Fanuc TP program (LS listing): hs_ov_h80_gutr.ls

/PROG  hs_ov_h80_gutr
/ATTR
COMMENT	= "19-03-05 13:35:50";
PROG_SIZE	= 0;
DEFAULT_GROUP	= 1, *, *, *, *;
/APPL
    ARC Welding Equipment: 1, *, *, *, *;
/MN
   1:  CALL HOME_ALL;
   1:  UFRAME_NUM = 1;
   1:  UTOOL_NUM = 3;
   1:  COL GUARD ADJUST 150;
   1:  PR[91] = PR[90];
   1:  PR[91,1] = PR[90,1] + 2.077;
   1:  PR[91,2] = PR[90,2] + 1.178;
   1:  PR[91,3] = PR[90,3] + 1.495;
   1:  PR[92] = PR[91];
   1:  PR[92,3] = PR[92,3] + 50;
   1:J PR[92] 10% FINE;
   1:L PR[91] R[100]mm/sec CNT100;
   1:  CALL LASER_DRAHT_START;
   1:  PR[91,1] = PR[90,1] + -2.557;
   1:L PR[91] R[100]mm/sec CNT100;
   1:  PR[91,1] = PR[90,1] + -4.760;
   1:  PR[91,2] = PR[90,2] + 1.925;
   1:L PR[91] R[100]mm/sec CNT100;
   1:  PR[91,1] = PR[90,1] + -5.957;
   1:  PR[91,2] = PR[90,2] + 3.712;
   1:L PR[91] R[100]mm/sec CNT100;
   1:  PR[91,1] = PR[90,1] + -7.859;
   1:  PR[91,2] = PR[90,2] + 8.118;
   1:L PR[91] R[100]mm/sec CNT100;
   1:  PR[91,1] = PR[90,1] + -8.020;
   1:  PR[91,2] = PR[90,2] + 8.503;
   1:L PR[91] R[100]mm/sec CNT100;
   1:  PR[91,1] = PR[90,1] + -8.141;
   1:  PR[91,2] = PR[90,2] + 8.842;
   1:L PR[91] R[100]mm/sec CNT100;
   1:  PR[91,1] = PR[90,1] + -8.162;
   1:  PR[91,2] = PR[90,2] + 8.883;
   1:L PR[91] R[100]mm/sec CNT100;
   1:  PR[91,1] = PR[90,1] + -11.179;
   1:  PR[91,2] = PR[90,2] + 12.501;
   1:L PR[91] R[100]mm/sec CNT100;
   1:  PR[91,1] = PR[90,1] + -11.400;
   1:  PR[91,2] = PR[90,2] + 12.803;
   1:L PR[91] R[100]mm/sec CNT100;
   1:  PR[91,1] = PR[90,1] + -11.431;
   1:  PR[91,2] = PR[90,2] + 12.835;
   1:L PR[91] R[100]mm/sec CNT100;
   1:  PR[91,1] = PR[90,1] + -15.350;
   1:  PR[91,2] = PR[90,2] + 15.448;
   1:L PR[91] R[100]mm/sec CNT100;
   1:  PR[91,1] = PR[90,1] + -15.648;
   1:  PR[91,2] = PR[90,2] + 15.676;
   1:L PR[91] R[100]mm/sec CNT100;
   1:  PR[91,1] = PR[90,1] + -15.686;
   1:  PR[91,2] = PR[90,2] + 15.697;
   1:L PR[91] R[100]mm/sec CNT100;
   1:  PR[91,1] = PR[90,1] + -20.186;
   1:  PR[91,2] = PR[90,2] + 17.090;
   1:L PR[91] R[100]mm/sec CNT100;
   1:  PR[91,1] = PR[90,1] + -20.537;
   1:  PR[91,2] = PR[90,2] + 17.225;
   1:L PR[91] R[100]mm/sec CNT100;
   1:  PR[91,1] = PR[90,1] + -20.579;
   1:  PR[91,2] = PR[90,2] + 17.235;
   1:L PR[91] R[100]mm/sec CNT100;
   1:  PR[91,1] = PR[90,1] + -25.291;
   1:  PR[91,2] = PR[90,2] + 17.293;
   1:L PR[91] R[100]mm/sec CNT100;
   1:  PR[91,1] = PR[90,1] + -25.667;
   1:  PR[91,2] = PR[90,2] + 17.323;
   1:L PR[91] R[100]mm/sec CNT100;
   1:  PR[91,1] = PR[90,1] + -25.709;
   1:  PR[91,2] = PR[90,2] + 17.320;
   1:L PR[91] R[100]mm/sec CNT100;
   1:  PR[91,1] = PR[90,1] + -30.244;
   1:  PR[91,2] = PR[90,2] + 16.038;
   1:L PR[91] R[100]mm/sec CNT100;
   1:  PR[91,1] = PR[90,1] + -30.614;
   1:  PR[91,2] = PR[90,2] + 15.960;
   1:L PR[91] R[100]mm/sec CNT100;
   1:  PR[91,1] = PR[90,1] + -30.652;
   1:  PR[91,2] = PR[90,2] + 15.946;
   1:L PR[91] R[100]mm/sec CNT100;
   1:  PR[91,1] = PR[90,1] + -34.635;
   1:  PR[91,2] = PR[90,2] + 13.430;
   1:L PR[91] R[100]mm/sec CNT100;
   1:  PR[91,1] = PR[90,1] + -34.968;
   1:  PR[91,2] = PR[90,2] + 13.250;
   1:L PR[91] R[100]mm/sec CNT100;
   1:  PR[91,1] = PR[90,1] + -35.000;
   1:  PR[91,2] = PR[90,2] + 13.227;
   1:L PR[91] R[100]mm/sec CNT100;
   1:  PR[91,1] = PR[90,1] + -38.105;
   1:  PR[91,2] = PR[90,2] + 9.684;
   1:L PR[91] R[100]mm/sec CNT100;
   1:  PR[91,1] = PR[90,1] + -38.375;
   1:  PR[91,2] = PR[90,2] + 9.416;
   1:L PR[91] R[100]mm/sec CNT100;
   1:  PR[91,1] = PR[90,1] + -38.398;
   1:  PR[91,2] = PR[90,2] + 9.386;
   1:L PR[91] R[100]mm/sec CNT100;
   1:  PR[91,1] = PR[90,1] + -40.370;
   1:  PR[91,2] = PR[90,2] + 5.107;
   1:L PR[91] R[100]mm/sec CNT100;
   1:  PR[91,1] = PR[90,1] + -40.554;
   1:  PR[91,2] = PR[90,2] + 4.773;
   1:L PR[91] R[100]mm/sec CNT100;
   1:  PR[91,1] = PR[90,1] + -40.567;
   1:  PR[91,2] = PR[90,2] + 4.738;
   1:L PR[91] R[100]mm/sec CNT100;
   1:  PR[91,1] = PR[90,1] + -41.243;
   1:  PR[91,2] = PR[90,2] + 0.073;
   1:L PR[91] R[100]mm/sec CNT100;
   1:  PR[91,1] = PR[90,1] + -41.325;
   1:  PR[91,2] = PR[90,2] + -0.300;
   1:L PR[91] R[100]mm/sec CNT100;
   1:  PR[91,1] = PR[90,1] + -41.327;
   1:  PR[91,2] = PR[90,2] + -0.336;
   1:L PR[91] R[100]mm/sec CNT100;
   1:  PR[91,1] = PR[90,1] + -40.651;
   1:  PR[91,2] = PR[90,2] + -5.001;
   1:L PR[91] R[100]mm/sec CNT100;
   1:  PR[91,1] = PR[90,1] + -40.624;
   1:  PR[91,2] = PR[90,2] + -5.383;
   1:L PR[91] R[100]mm/sec CNT100;
   1:  PR[91,1] = PR[90,1] + -40.597;
   1:  PR[91,2] = PR[90,2] + -5.504;
   1:L PR[91] R[100]mm/sec CNT100;
   1:  PR[91,1] = PR[90,1] + -40.524;
   1:  PR[91,2] = PR[90,2] + -5.699;
   1:L PR[91] R[100]mm/sec CNT100;
   1:  PR[91,1] = PR[90,1] + -38.552;
   1:  PR[91,2] = PR[90,2] + -9.979;
   1:L PR[91] R[100]mm/sec CNT100;
   1:  PR[91,1] = PR[90,1] + -38.450;
   1:  PR[91,2] = PR[90,2] + -10.165;
   1:L PR[91] R[100]mm/sec CNT100;
   1:  PR[91,1] = PR[90,1] + -38.325;
   1:  PR[91,2] = PR[90,2] + -10.331;
   1:L PR[91] R[100]mm/sec CNT100;
   1:  PR[91,1] = PR[90,1] + -35.219;
   1:  PR[91,2] = PR[90,2] + -13.874;
   1:L PR[91] R[100]mm/sec CNT100;
   1:  PR[91,1] = PR[90,1] + -35.068;
   1:  PR[91,2] = PR[90,2] + -14.024;
   1:L PR[91] R[100]mm/sec CNT100;
   1:  PR[91,1] = PR[90,1] + -34.902;
   1:  PR[91,2] = PR[90,2] + -14.147;
   1:L PR[91] R[100]mm/sec CNT100;
   1:  PR[91,1] = PR[90,1] + -30.918;
   1:  PR[91,2] = PR[90,2] + -16.664;
   1:L PR[91] R[100]mm/sec CNT100;
   1:  PR[91,1] = PR[90,1] + -30.730;
   1:  PR[91,2] = PR[90,2] + -16.765;
   1:L PR[91] R[100]mm/sec CNT100;
   1:  PR[91,1] = PR[90,1] + -30.537;
   1:  PR[91,2] = PR[90,2] + -16.836;
   1:L PR[91] R[100]mm/sec CNT100;
   1:  PR[91,1] = PR[90,1] + -26.001;
   1:  PR[91,2] = PR[90,2] + -18.118;
   1:L PR[91] R[100]mm/sec CNT100;
   1:  PR[91,1] = PR[90,1] + -25.791;
   1:  PR[91,2] = PR[90,2] + -18.162;
   1:L PR[91] R[100]mm/sec CNT100;
   1:  PR[91,1] = PR[90,1] + -25.587;
   1:  PR[91,2] = PR[90,2] + -18.175;
   1:L PR[91] R[100]mm/sec CNT100;
   1:  PR[91,1] = PR[90,1] + -20.873;
   1:  PR[91,2] = PR[90,2] + -18.117;
   1:L PR[91] R[100]mm/sec CNT100;
   1:  PR[91,1] = PR[90,1] + -20.658;
   1:  PR[91,2] = PR[90,2] + -18.100;
   1:L PR[91] R[100]mm/sec CNT100;
   1:  PR[91,1] = PR[90,1] + -20.460;
   1:  PR[91,2] = PR[90,2] + -18.055;
   1:L PR[91] R[100]mm/sec CNT100;
   1:  PR[91,1] = PR[90,1] + -15.959;
   1:  PR[91,2] = PR[90,2] + -16.661;
   1:L PR[91] R[100]mm/sec CNT100;
   1:  PR[91,1] = PR[90,1] + -15.756;
   1:  PR[91,2] = PR[90,2] + -16.583;
   1:L PR[91] R[100]mm/sec CNT100;
   1:  PR[91,1] = PR[90,1] + -15.579;
   1:  PR[91,2] = PR[90,2] + -16.484;
   1:L PR[91] R[100]mm/sec CNT100;
   1:  PR[91,1] = PR[90,1] + -11.659;
   1:  PR[91,2] = PR[90,2] + -13.871;
   1:L PR[91] R[100]mm/sec CNT100;
   1:  PR[91,1] = PR[90,1] + -11.486;
   1:  PR[91,2] = PR[90,2] + -13.739;
   1:L PR[91] R[100]mm/sec CNT100;
   1:  PR[91,1] = PR[90,1] + -11.345;
   1:  PR[91,2] = PR[90,2] + -13.595;
   1:L PR[91] R[100]mm/sec CNT100;
   1:  PR[91,1] = PR[90,1] + -8.328;
   1:  PR[91,2] = PR[90,2] + -9.976;
   1:L PR[91] R[100]mm/sec CNT100;
   1:  PR[91,1] = PR[90,1] + -8.199;
   1:  PR[91,2] = PR[90,2] + -9.799;
   1:L PR[91] R[100]mm/sec CNT100;
   1:  PR[91,1] = PR[90,1] + -8.105;
   1:  PR[91,2] = PR[90,2] + -9.621;
   1:L PR[91] R[100]mm/sec CNT100;
   1:  PR[91,1] = PR[90,1] + -6.242;
   1:  PR[91,2] = PR[90,2] + -5.303;
   1:L PR[91] R[100]mm/sec CNT100;
   1:  PR[91,1] = PR[90,1] + -6.003;
   1:  PR[91,2] = PR[90,2] + -4.628;
   1:L PR[91] R[100]mm/sec CNT100;
   1:  PR[91,1] = PR[90,1] + -4.760;
   1:  PR[91,2] = PR[90,2] + -2.773;
   1:L PR[91] R[100]mm/sec CNT100;
   1:  PR[91,1] = PR[90,1] + -2.557;
   1:  PR[91,2] = PR[90,2] + -2.026;
   1:L PR[91] R[100]mm/sec CNT100;
   1:  PR[91,1] = PR[90,1] + 2.077;
   1:L PR[91] R[100]mm/sec CNT100;
   1:  PR[91,1] = PR[90,1] + 4.281;
   1:  PR[91,2] = PR[90,2] + -2.773;
   1:L PR[91] R[100]mm/sec CNT100;
   1:  PR[91,1] = PR[90,1] + 5.478;
   1:  PR[91,2] = PR[90,2] + -4.559;
   1:L PR[91] R[100]mm/sec CNT100;
   1:  PR[91,1] = PR[90,1] + 7.379;
   1:  PR[91,2] = PR[90,2] + -8.965;
   1:L PR[91] R[100]mm/sec CNT100;
   1:  PR[91,1] = PR[90,1] + 7.540;
   1:  PR[91,2] = PR[90,2] + -9.350;
   1:L PR[91] R[100]mm/sec CNT100;
   1:  PR[91,1] = PR[90,1] + 7.661;
   1:  PR[91,2] = PR[90,2] + -9.690;
   1:L PR[91] R[100]mm/sec CNT100;
   1:  PR[91,1] = PR[90,1] + 7.683;
   1:  PR[91,2] = PR[90,2] + -9.730;
   1:L PR[91] R[100]mm/sec CNT100;
   1:  PR[91,1] = PR[90,1] + 10.700;
   1:  PR[91,2] = PR[90,2] + -13.348;
   1:L PR[91] R[100]mm/sec CNT100;
   1:  PR[91,1] = PR[90,1] + 10.920;
   1:  PR[91,2] = PR[90,2] + -13.650;
   1:L PR[91] R[100]mm/sec CNT100;
   1:  PR[91,1] = PR[90,1] + 10.951;
   1:  PR[91,2] = PR[90,2] + -13.682;
   1:L PR[91] R[100]mm/sec CNT100;
   1:  PR[91,1] = PR[90,1] + 14.871;
   1:  PR[91,2] = PR[90,2] + -16.295;
   1:L PR[91] R[100]mm/sec CNT100;
   1:  PR[91,1] = PR[90,1] + 15.168;
   1:  PR[91,2] = PR[90,2] + -16.523;
   1:L PR[91] R[100]mm/sec CNT100;
   1:  PR[91,1] = PR[90,1] + 15.207;
   1:  PR[91,2] = PR[90,2] + -16.544;
   1:L PR[91] R[100]mm/sec CNT100;
   1:  PR[91,1] = PR[90,1] + 19.707;
   1:  PR[91,2] = PR[90,2] + -17.938;
   1:L PR[91] R[100]mm/sec CNT100;
   1:  PR[91,1] = PR[90,1] + 20.058;
   1:  PR[91,2] = PR[90,2] + -18.072;
   1:L PR[91] R[100]mm/sec CNT100;
   1:  PR[91,1] = PR[90,1] + 20.099;
   1:  PR[91,2] = PR[90,2] + -18.082;
   1:L PR[91] R[100]mm/sec CNT100;
   1:  PR[91,1] = PR[90,1] + 24.812;
   1:  PR[91,2] = PR[90,2] + -18.140;
   1:L PR[91] R[100]mm/sec CNT100;
   1:  PR[91,1] = PR[90,1] + 25.187;
   1:  PR[91,2] = PR[90,2] + -18.170;
   1:L PR[91] R[100]mm/sec CNT100;
   1:  PR[91,1] = PR[90,1] + 25.229;
   1:  PR[91,2] = PR[90,2] + -18.168;
   1:L PR[91] R[100]mm/sec CNT100;
   1:  PR[91,1] = PR[90,1] + 29.764;
   1:  PR[91,2] = PR[90,2] + -16.885;
   1:L PR[91] R[100]mm/sec CNT100;
   1:  PR[91,1] = PR[90,1] + 30.134;
   1:  PR[91,2] = PR[90,2] + -16.808;
   1:L PR[91] R[100]mm/sec CNT100;
   1:  PR[91,1] = PR[90,1] + 30.172;
   1:  PR[91,2] = PR[90,2] + -16.794;
   1:L PR[91] R[100]mm/sec CNT100;
   1:  PR[91,1] = PR[90,1] + 34.155;
   1:  PR[91,2] = PR[90,2] + -14.277;
   1:L PR[91] R[100]mm/sec CNT100;
   1:  PR[91,1] = PR[90,1] + 34.489;
   1:  PR[91,2] = PR[90,2] + -14.098;
   1:L PR[91] R[100]mm/sec CNT100;
   1:  PR[91,1] = PR[90,1] + 34.521;
   1:  PR[91,2] = PR[90,2] + -14.074;
   1:L PR[91] R[100]mm/sec CNT100;
   1:  PR[91,1] = PR[90,1] + 37.626;
   1:  PR[91,2] = PR[90,2] + -10.531;
   1:L PR[91] R[100]mm/sec CNT100;
   1:  PR[91,1] = PR[90,1] + 37.895;
   1:  PR[91,2] = PR[90,2] + -10.264;
   1:L PR[91] R[100]mm/sec CNT100;
   1:  PR[91,1] = PR[90,1] + 37.919;
   1:  PR[91,2] = PR[90,2] + -10.233;
   1:L PR[91] R[100]mm/sec CNT100;
   1:  PR[91,1] = PR[90,1] + 39.891;
   1:  PR[91,2] = PR[90,2] + -5.954;
   1:L PR[91] R[100]mm/sec CNT100;
   1:  PR[91,1] = PR[90,1] + 40.074;
   1:  PR[91,2] = PR[90,2] + -5.620;
   1:L PR[91] R[100]mm/sec CNT100;
   1:  PR[91,1] = PR[90,1] + 40.087;
   1:  PR[91,2] = PR[90,2] + -5.585;
   1:L PR[91] R[100]mm/sec CNT100;
   1:  PR[91,1] = PR[90,1] + 40.764;
   1:  PR[91,2] = PR[90,2] + -0.920;
   1:L PR[91] R[100]mm/sec CNT100;
   1:  PR[91,1] = PR[90,1] + 40.845;
   1:  PR[91,2] = PR[90,2] + -0.547;
   1:L PR[91] R[100]mm/sec CNT100;
   1:  PR[91,1] = PR[90,1] + 40.848;
   1:  PR[91,2] = PR[90,2] + -0.511;
   1:L PR[91] R[100]mm/sec CNT100;
   1:  PR[91,1] = PR[90,1] + 40.171;
   1:  PR[91,2] = PR[90,2] + 4.154;
   1:L PR[91] R[100]mm/sec CNT100;
   1:  PR[91,1] = PR[90,1] + 40.144;
   1:  PR[91,2] = PR[90,2] + 4.536;
   1:L PR[91] R[100]mm/sec CNT100;
   1:  PR[91,1] = PR[90,1] + 40.117;
   1:  PR[91,2] = PR[90,2] + 4.657;
   1:L PR[91] R[100]mm/sec CNT100;
   1:  PR[91,1] = PR[90,1] + 40.044;
   1:  PR[91,2] = PR[90,2] + 4.852;
   1:L PR[91] R[100]mm/sec CNT100;
   1:  PR[91,1] = PR[90,1] + 38.072;
   1:  PR[91,2] = PR[90,2] + 9.132;
   1:L PR[91] R[100]mm/sec CNT100;
   1:  PR[91,1] = PR[90,1] + 37.970;
   1:  PR[91,2] = PR[90,2] + 9.318;
   1:L PR[91] R[100]mm/sec CNT100;
   1:  PR[91,1] = PR[90,1] + 37.845;
   1:  PR[91,2] = PR[90,2] + 9.483;
   1:L PR[91] R[100]mm/sec CNT100;
   1:  PR[91,1] = PR[90,1] + 34.739;
   1:  PR[91,2] = PR[90,2] + 13.027;
   1:L PR[91] R[100]mm/sec CNT100;
   1:  PR[91,1] = PR[90,1] + 34.588;
   1:  PR[91,2] = PR[90,2] + 13.177;
   1:L PR[91] R[100]mm/sec CNT100;
   1:  PR[91,1] = PR[90,1] + 34.422;
   1:  PR[91,2] = PR[90,2] + 13.300;
   1:L PR[91] R[100]mm/sec CNT100;
   1:  PR[91,1] = PR[90,1] + 30.438;
   1:  PR[91,2] = PR[90,2] + 15.816;
   1:L PR[91] R[100]mm/sec CNT100;
   1:  PR[91,1] = PR[90,1] + 30.250;
   1:  PR[91,2] = PR[90,2] + 15.918;
   1:L PR[91] R[100]mm/sec CNT100;
   1:  PR[91,1] = PR[90,1] + 30.057;
   1:  PR[91,2] = PR[90,2] + 15.988;
   1:L PR[91] R[100]mm/sec CNT100;
   1:  PR[91,1] = PR[90,1] + 25.521;
   1:  PR[91,2] = PR[90,2] + 17.271;
   1:L PR[91] R[100]mm/sec CNT100;
   1:  PR[91,1] = PR[90,1] + 25.311;
   1:  PR[91,2] = PR[90,2] + 17.315;
   1:L PR[91] R[100]mm/sec CNT100;
   1:  PR[91,1] = PR[90,1] + 25.107;
   1:  PR[91,2] = PR[90,2] + 17.328;
   1:L PR[91] R[100]mm/sec CNT100;
   1:  PR[91,1] = PR[90,1] + 20.394;
   1:  PR[91,2] = PR[90,2] + 17.270;
   1:L PR[91] R[100]mm/sec CNT100;
   1:  PR[91,1] = PR[90,1] + 20.178;
   1:  PR[91,2] = PR[90,2] + 17.253;
   1:L PR[91] R[100]mm/sec CNT100;
   1:  PR[91,1] = PR[90,1] + 19.980;
   1:  PR[91,2] = PR[90,2] + 17.207;
   1:L PR[91] R[100]mm/sec CNT100;
   1:  PR[91,1] = PR[90,1] + 15.479;
   1:  PR[91,2] = PR[90,2] + 15.814;
   1:L PR[91] R[100]mm/sec CNT100;
   1:  PR[91,1] = PR[90,1] + 15.276;
   1:  PR[91,2] = PR[90,2] + 15.736;
   1:L PR[91] R[100]mm/sec CNT100;
   1:  PR[91,1] = PR[90,1] + 15.100;
   1:  PR[91,2] = PR[90,2] + 15.637;
   1:L PR[91] R[100]mm/sec CNT100;
   1:  PR[91,1] = PR[90,1] + 11.180;
   1:  PR[91,2] = PR[90,2] + 13.024;
   1:L PR[91] R[100]mm/sec CNT100;
   1:  PR[91,1] = PR[90,1] + 11.007;
   1:  PR[91,2] = PR[90,2] + 12.892;
   1:L PR[91] R[100]mm/sec CNT100;
   1:  PR[91,1] = PR[90,1] + 10.866;
   1:  PR[91,2] = PR[90,2] + 12.747;
   1:L PR[91] R[100]mm/sec CNT100;
   1:  PR[91,1] = PR[90,1] + 7.848;
   1:  PR[91,2] = PR[90,2] + 9.129;
   1:L PR[91] R[100]mm/sec CNT100;
   1:  PR[91,1] = PR[90,1] + 7.719;
   1:  PR[91,2] = PR[90,2] + 8.952;
   1:L PR[91] R[100]mm/sec CNT100;
   1:  PR[91,1] = PR[90,1] + 7.625;
   1:  PR[91,2] = PR[90,2] + 8.774;
   1:L PR[91] R[100]mm/sec CNT100;
   1:  PR[91,1] = PR[90,1] + 5.762;
   1:  PR[91,2] = PR[90,2] + 4.456;
   1:L PR[91] R[100]mm/sec CNT100;
   1:  PR[91,1] = PR[90,1] + 5.524;
   1:  PR[91,2] = PR[90,2] + 3.781;
   1:L PR[91] R[100]mm/sec CNT100;
   1:  PR[91,1] = PR[90,1] + 4.281;
   1:  PR[91,2] = PR[90,2] + 1.925;
   1:L PR[91] R[100]mm/sec CNT100;
   1:  PR[91,1] = PR[90,1] + 2.077;
   1:  PR[91,2] = PR[90,2] + 1.178;
   1:L PR[91] R[100]mm/sec CNT100;
   1:  PR[91] = PR[90];
   1:  PR[91,1] = PR[90,1] + -2.557;
   1:  PR[91,3] = PR[90,3] + 2.795;
   1:L PR[91] R[100]mm/sec CNT100;
   1:  PR[91,1] = PR[90,1] + -4.760;
   1:  PR[91,2] = PR[90,2] + 1.925;
   1:L PR[91] R[100]mm/sec CNT100;
   1:  PR[91,1] = PR[90,1] + -5.959;
   1:  PR[91,2] = PR[90,2] + 3.715;
   1:L PR[91] R[100]mm/sec CNT100;
   1:  PR[91,1] = PR[90,1] + -7.336;
   1:  PR[91,2] = PR[90,2] + 6.933;
   1:L PR[91] R[100]mm/sec CNT100;
   1:  PR[91,1] = PR[90,1] + -7.755;
   1:  PR[91,2] = PR[90,2] + 8.106;
   1:L PR[91] R[100]mm/sec CNT100;
   1:  PR[91,1] = PR[90,1] + -8.186;
   1:  PR[91,2] = PR[90,2] + 8.922;
   1:L PR[91] R[100]mm/sec CNT100;
   1:  PR[91,1] = PR[90,1] + -10.080;
   1:  PR[91,2] = PR[90,2] + 11.193;
   1:L PR[91] R[100]mm/sec CNT100;
   1:  PR[91,1] = PR[90,1] + -10.818;
   1:  PR[91,2] = PR[90,2] + 12.203;
   1:L PR[91] R[100]mm/sec CNT100;
   1:  PR[91,1] = PR[90,1] + -11.462;
   1:  PR[91,2] = PR[90,2] + 12.862;
   1:L PR[91] R[100]mm/sec CNT100;
   1:  PR[91,1] = PR[90,1] + -13.922;
   1:  PR[91,2] = PR[90,2] + 14.503;
   1:L PR[91] R[100]mm/sec CNT100;
   1:  PR[91,1] = PR[90,1] + -14.916;
   1:  PR[91,2] = PR[90,2] + 15.263;
   1:L PR[91] R[100]mm/sec CNT100;
   1:  PR[91,1] = PR[90,1] + -15.719;
   1:  PR[91,2] = PR[90,2] + 15.713;
   1:L PR[91] R[100]mm/sec CNT100;
   1:  PR[91,1] = PR[90,1] + -18.544;
   1:  PR[91,2] = PR[90,2] + 16.587;
   1:L PR[91] R[100]mm/sec CNT100;
   1:  PR[91,1] = PR[90,1] + -19.713;
   1:  PR[91,2] = PR[90,2] + 17.036;
   1:L PR[91] R[100]mm/sec CNT100;
   1:  PR[91,1] = PR[90,1] + -20.610;
   1:  PR[91,2] = PR[90,2] + 17.239;
   1:L PR[91] R[100]mm/sec CNT100;
   1:  PR[91,1] = PR[90,1] + -23.569;
   1:  PR[91,2] = PR[90,2] + 17.276;
   1:L PR[91] R[100]mm/sec CNT100;
   1:  PR[91,1] = PR[90,1] + -24.818;
   1:  PR[91,2] = PR[90,2] + 17.376;
   1:L PR[91] R[100]mm/sec CNT100;
   1:  PR[91,1] = PR[90,1] + -25.734;
   1:  PR[91,2] = PR[90,2] + 17.317;
   1:L PR[91] R[100]mm/sec CNT100;
   1:  PR[91,1] = PR[90,1] + -28.581;
   1:  PR[91,2] = PR[90,2] + 16.512;
   1:L PR[91] R[100]mm/sec CNT100;
   1:  PR[91,1] = PR[90,1] + -29.809;
   1:  PR[91,2] = PR[90,2] + 16.253;
   1:L PR[91] R[100]mm/sec CNT100;
   1:  PR[91,1] = PR[90,1] + -30.670;
   1:  PR[91,2] = PR[90,2] + 15.938;
   1:L PR[91] R[100]mm/sec CNT100;
   1:  PR[91,1] = PR[90,1] + -33.171;
   1:  PR[91,2] = PR[90,2] + 14.358;
   1:L PR[91] R[100]mm/sec CNT100;
   1:  PR[91,1] = PR[90,1] + -34.276;
   1:  PR[91,2] = PR[90,2] + 13.762;
   1:L PR[91] R[100]mm/sec CNT100;
   1:  PR[91,1] = PR[90,1] + -35.012;
   1:  PR[91,2] = PR[90,2] + 13.217;
   1:L PR[91] R[100]mm/sec CNT100;
   1:  PR[91,1] = PR[90,1] + -36.961;
   1:  PR[91,2] = PR[90,2] + 10.993;
   1:L PR[91] R[100]mm/sec CNT100;
   1:  PR[91,1] = PR[90,1] + -37.853;
   1:  PR[91,2] = PR[90,2] + 10.108;
   1:L PR[91] R[100]mm/sec CNT100;
   1:  PR[91,1] = PR[90,1] + -38.404;
   1:  PR[91,2] = PR[90,2] + 9.377;
   1:L PR[91] R[100]mm/sec CNT100;
   1:  PR[91,1] = PR[90,1] + -39.642;
   1:  PR[91,2] = PR[90,2] + 6.690;
   1:L PR[91] R[100]mm/sec CNT100;
   1:  PR[91,1] = PR[90,1] + -40.248;
   1:  PR[91,2] = PR[90,2] + 5.588;
   1:L PR[91] R[100]mm/sec CNT100;
   1:  PR[91,1] = PR[90,1] + -40.569;
   1:  PR[91,2] = PR[90,2] + 4.732;
   1:L PR[91] R[100]mm/sec CNT100;
   1:  PR[91,1] = PR[90,1] + -40.993;
   1:  PR[91,2] = PR[90,2] + 1.804;
   1:L PR[91] R[100]mm/sec CNT100;
   1:  PR[91,1] = PR[90,1] + -41.262;
   1:  PR[91,2] = PR[90,2] + 0.574;
   1:L PR[91] R[100]mm/sec CNT100;
   1:  PR[91,1] = PR[90,1] + -41.327;
   1:  PR[91,2] = PR[90,2] + -0.336;
   1:L PR[91] R[100]mm/sec CNT100;
   1:  PR[91,1] = PR[90,1] + -40.903;
   1:  PR[91,2] = PR[90,2] + -3.265;
   1:L PR[91] R[100]mm/sec CNT100;
   1:  PR[91,1] = PR[90,1] + -40.812;
   1:  PR[91,2] = PR[90,2] + -4.521;
   1:L PR[91] R[100]mm/sec CNT100;
   1:  PR[91,1] = PR[90,1] + -40.599;
   1:  PR[91,2] = PR[90,2] + -5.499;
   1:L PR[91] R[100]mm/sec CNT100;
   1:  PR[91,1] = PR[90,1] + -40.218;
   1:  PR[91,2] = PR[90,2] + -6.515;
   1:L PR[91] R[100]mm/sec CNT100;
   1:  PR[91,1] = PR[90,1] + -38.979;
   1:  PR[91,2] = PR[90,2] + -9.202;
   1:L PR[91] R[100]mm/sec CNT100;
   1:  PR[91,1] = PR[90,1] + -38.455;
   1:  PR[91,2] = PR[90,2] + -10.156;
   1:L PR[91] R[100]mm/sec CNT100;
   1:  PR[91,1] = PR[90,1] + -37.803;
   1:  PR[91,2] = PR[90,2] + -11.022;
   1:L PR[91] R[100]mm/sec CNT100;
   1:  PR[91,1] = PR[90,1] + -35.853;
   1:  PR[91,2] = PR[90,2] + -13.246;
   1:L PR[91] R[100]mm/sec CNT100;
   1:  PR[91,1] = PR[90,1] + -35.080;
   1:  PR[91,2] = PR[90,2] + -14.014;
   1:L PR[91] R[100]mm/sec CNT100;
   1:  PR[91,1] = PR[90,1] + -34.210;
   1:  PR[91,2] = PR[90,2] + -14.659;
   1:L PR[91] R[100]mm/sec CNT100;
   1:  PR[91,1] = PR[90,1] + -31.708;
   1:  PR[91,2] = PR[90,2] + -16.239;
   1:L PR[91] R[100]mm/sec CNT100;
   1:  PR[91,1] = PR[90,1] + -30.749;
   1:  PR[91,2] = PR[90,2] + -16.757;
   1:L PR[91] R[100]mm/sec CNT100;
   1:  PR[91,1] = PR[90,1] + -29.732;
   1:  PR[91,2] = PR[90,2] + -17.129;
   1:L PR[91] R[100]mm/sec CNT100;
   1:  PR[91,1] = PR[90,1] + -26.884;
   1:  PR[91,2] = PR[90,2] + -17.934;
   1:L PR[91] R[100]mm/sec CNT100;
   1:  PR[91,1] = PR[90,1] + -25.817;
   1:  PR[91,2] = PR[90,2] + -18.159;
   1:L PR[91] R[100]mm/sec CNT100;
   1:  PR[91,1] = PR[90,1] + -24.738;
   1:  PR[91,2] = PR[90,2] + -18.228;
   1:L PR[91] R[100]mm/sec CNT100;
   1:  PR[91,1] = PR[90,1] + -21.778;
   1:  PR[91,2] = PR[90,2] + -18.191;
   1:L PR[91] R[100]mm/sec CNT100;
   1:  PR[91,1] = PR[90,1] + -20.689;
   1:  PR[91,2] = PR[90,2] + -18.105;
   1:L PR[91] R[100]mm/sec CNT100;
   1:  PR[91,1] = PR[90,1] + -19.636;
   1:  PR[91,2] = PR[90,2] + -17.866;
   1:L PR[91] R[100]mm/sec CNT100;
   1:  PR[91,1] = PR[90,1] + -16.810;
   1:  PR[91,2] = PR[90,2] + -16.991;
   1:L PR[91] R[100]mm/sec CNT100;
   1:  PR[91,1] = PR[90,1] + -15.789;
   1:  PR[91,2] = PR[90,2] + -16.599;
   1:L PR[91] R[100]mm/sec CNT100;
   1:  PR[91,1] = PR[90,1] + -14.847;
   1:  PR[91,2] = PR[90,2] + -16.072;
   1:L PR[91] R[100]mm/sec CNT100;
   1:  PR[91,1] = PR[90,1] + -12.386;
   1:  PR[91,2] = PR[90,2] + -14.431;
   1:L PR[91] R[100]mm/sec CNT100;
   1:  PR[91,1] = PR[90,1] + -11.517;
   1:  PR[91,2] = PR[90,2] + -13.766;
   1:L PR[91] R[100]mm/sec CNT100;
   1:  PR[91,1] = PR[90,1] + -10.763;
   1:  PR[91,2] = PR[90,2] + -12.995;
   1:L PR[91] R[100]mm/sec CNT100;
   1:  PR[91,1] = PR[90,1] + -8.869;
   1:  PR[91,2] = PR[90,2] + -10.723;
   1:L PR[91] R[100]mm/sec CNT100;
   1:  PR[91,1] = PR[90,1] + -8.223;
   1:  PR[91,2] = PR[90,2] + -9.838;
   1:L PR[91] R[100]mm/sec CNT100;
   1:  PR[91,1] = PR[90,1] + -7.719;
   1:  PR[91,2] = PR[90,2] + -8.886;
   1:L PR[91] R[100]mm/sec CNT100;
   1:  PR[91,1] = PR[90,1] + -6.550;
   1:  PR[91,2] = PR[90,2] + -6.176;
   1:L PR[91] R[100]mm/sec CNT100;
   1:  PR[91,1] = PR[90,1] + -6.003;
   1:  PR[91,2] = PR[90,2] + -4.628;
   1:L PR[91] R[100]mm/sec CNT100;
   1:  PR[91,1] = PR[90,1] + -4.760;
   1:  PR[91,2] = PR[90,2] + -2.773;
   1:L PR[91] R[100]mm/sec CNT100;
   1:  PR[91,1] = PR[90,1] + -2.557;
   1:  PR[91,2] = PR[90,2] + -2.026;
   1:L PR[91] R[100]mm/sec CNT100;
   1:  PR[91,1] = PR[90,1] + 2.077;
   1:L PR[91] R[100]mm/sec CNT100;
   1:  PR[91,1] = PR[90,1] + 4.280;
   1:  PR[91,2] = PR[90,2] + -2.773;
   1:L PR[91] R[100]mm/sec CNT100;
   1:  PR[91,1] = PR[90,1] + 5.480;
   1:  PR[91,2] = PR[90,2] + -4.563;
   1:L PR[91] R[100]mm/sec CNT100;
   1:  PR[91,1] = PR[90,1] + 6.856;
   1:  PR[91,2] = PR[90,2] + -7.781;
   1:L PR[91] R[100]mm/sec CNT100;
   1:  PR[91,1] = PR[90,1] + 7.275;
   1:  PR[91,2] = PR[90,2] + -8.954;
   1:L PR[91] R[100]mm/sec CNT100;
   1:  PR[91,1] = PR[90,1] + 7.707;
   1:  PR[91,2] = PR[90,2] + -9.769;
   1:L PR[91] R[100]mm/sec CNT100;
   1:  PR[91,1] = PR[90,1] + 9.601;
   1:  PR[91,2] = PR[90,2] + -12.040;
   1:L PR[91] R[100]mm/sec CNT100;
   1:  PR[91,1] = PR[90,1] + 10.338;
   1:  PR[91,2] = PR[90,2] + -13.051;
   1:L PR[91] R[100]mm/sec CNT100;
   1:  PR[91,1] = PR[90,1] + 10.982;
   1:  PR[91,2] = PR[90,2] + -13.710;
   1:L PR[91] R[100]mm/sec CNT100;
   1:  PR[91,1] = PR[90,1] + 13.442;
   1:  PR[91,2] = PR[90,2] + -15.350;
   1:L PR[91] R[100]mm/sec CNT100;
   1:  PR[91,1] = PR[90,1] + 14.436;
   1:  PR[91,2] = PR[90,2] + -16.111;
   1:L PR[91] R[100]mm/sec CNT100;
   1:  PR[91,1] = PR[90,1] + 15.239;
   1:  PR[91,2] = PR[90,2] + -16.560;
   1:L PR[91] R[100]mm/sec CNT100;
   1:  PR[91,1] = PR[90,1] + 18.065;
   1:  PR[91,2] = PR[90,2] + -17.435;
   1:L PR[91] R[100]mm/sec CNT100;
   1:  PR[91,1] = PR[90,1] + 19.234;
   1:  PR[91,2] = PR[90,2] + -17.883;
   1:L PR[91] R[100]mm/sec CNT100;
   1:  PR[91,1] = PR[90,1] + 20.130;
   1:  PR[91,2] = PR[90,2] + -18.087;
   1:L PR[91] R[100]mm/sec CNT100;
   1:  PR[91,1] = PR[90,1] + 23.089;
   1:  PR[91,2] = PR[90,2] + -18.123;
   1:L PR[91] R[100]mm/sec CNT100;
   1:  PR[91,1] = PR[90,1] + 24.338;
   1:  PR[91,2] = PR[90,2] + -18.223;
   1:L PR[91] R[100]mm/sec CNT100;
   1:  PR[91,1] = PR[90,1] + 25.255;
   1:  PR[91,2] = PR[90,2] + -18.164;
   1:L PR[91] R[100]mm/sec CNT100;
   1:  PR[91,1] = PR[90,1] + 28.102;
   1:  PR[91,2] = PR[90,2] + -17.359;
   1:L PR[91] R[100]mm/sec CNT100;
   1:  PR[91,1] = PR[90,1] + 29.329;
   1:  PR[91,2] = PR[90,2] + -17.101;
   1:L PR[91] R[100]mm/sec CNT100;
   1:  PR[91,1] = PR[90,1] + 30.191;
   1:  PR[91,2] = PR[90,2] + -16.785;
   1:L PR[91] R[100]mm/sec CNT100;
   1:  PR[91,1] = PR[90,1] + 32.691;
   1:  PR[91,2] = PR[90,2] + -15.206;
   1:L PR[91] R[100]mm/sec CNT100;
   1:  PR[91,1] = PR[90,1] + 33.796;
   1:  PR[91,2] = PR[90,2] + -14.610;
   1:L PR[91] R[100]mm/sec CNT100;
   1:  PR[91,1] = PR[90,1] + 34.532;
   1:  PR[91,2] = PR[90,2] + -14.064;
   1:L PR[91] R[100]mm/sec CNT100;
   1:  PR[91,1] = PR[90,1] + 36.482;
   1:  PR[91,2] = PR[90,2] + -11.840;
   1:L PR[91] R[100]mm/sec CNT100;
   1:  PR[91,1] = PR[90,1] + 37.374;
   1:  PR[91,2] = PR[90,2] + -10.955;
   1:L PR[91] R[100]mm/sec CNT100;
   1:  PR[91,1] = PR[90,1] + 37.924;
   1:  PR[91,2] = PR[90,2] + -10.224;
   1:L PR[91] R[100]mm/sec CNT100;
   1:  PR[91,1] = PR[90,1] + 39.162;
   1:  PR[91,2] = PR[90,2] + -7.538;
   1:L PR[91] R[100]mm/sec CNT100;
   1:  PR[91,1] = PR[90,1] + 39.768;
   1:  PR[91,2] = PR[90,2] + -6.435;
   1:L PR[91] R[100]mm/sec CNT100;
   1:  PR[91,1] = PR[90,1] + 40.089;
   1:  PR[91,2] = PR[90,2] + -5.579;
   1:L PR[91] R[100]mm/sec CNT100;
   1:  PR[91,1] = PR[90,1] + 40.513;
   1:  PR[91,2] = PR[90,2] + -2.651;
   1:L PR[91] R[100]mm/sec CNT100;
   1:  PR[91,1] = PR[90,1] + 40.782;
   1:  PR[91,2] = PR[90,2] + -1.422;
   1:L PR[91] R[100]mm/sec CNT100;
   1:  PR[91,1] = PR[90,1] + 40.848;
   1:  PR[91,2] = PR[90,2] + -0.511;
   1:L PR[91] R[100]mm/sec CNT100;
   1:  PR[91,1] = PR[90,1] + 40.423;
   1:  PR[91,2] = PR[90,2] + 2.417;
   1:L PR[91] R[100]mm/sec CNT100;
   1:  PR[91,1] = PR[90,1] + 40.333;
   1:  PR[91,2] = PR[90,2] + 3.674;
   1:L PR[91] R[100]mm/sec CNT100;
   1:  PR[91,1] = PR[90,1] + 40.119;
   1:  PR[91,2] = PR[90,2] + 4.651;
   1:L PR[91] R[100]mm/sec CNT100;
   1:  PR[91,1] = PR[90,1] + 39.738;
   1:  PR[91,2] = PR[90,2] + 5.667;
   1:L PR[91] R[100]mm/sec CNT100;
   1:  PR[91,1] = PR[90,1] + 38.500;
   1:  PR[91,2] = PR[90,2] + 8.355;
   1:L PR[91] R[100]mm/sec CNT100;
   1:  PR[91,1] = PR[90,1] + 37.976;
   1:  PR[91,2] = PR[90,2] + 9.309;
   1:L PR[91] R[100]mm/sec CNT100;
   1:  PR[91,1] = PR[90,1] + 37.323;
   1:  PR[91,2] = PR[90,2] + 10.175;
   1:L PR[91] R[100]mm/sec CNT100;
   1:  PR[91,1] = PR[90,1] + 35.373;
   1:  PR[91,2] = PR[90,2] + 12.399;
   1:L PR[91] R[100]mm/sec CNT100;
   1:  PR[91,1] = PR[90,1] + 34.600;
   1:  PR[91,2] = PR[90,2] + 13.167;
   1:L PR[91] R[100]mm/sec CNT100;
   1:  PR[91,1] = PR[90,1] + 33.730;
   1:  PR[91,2] = PR[90,2] + 13.812;
   1:L PR[91] R[100]mm/sec CNT100;
   1:  PR[91,1] = PR[90,1] + 31.229;
   1:  PR[91,2] = PR[90,2] + 15.392;
   1:L PR[91] R[100]mm/sec CNT100;
   1:  PR[91,1] = PR[90,1] + 30.269;
   1:  PR[91,2] = PR[90,2] + 15.909;
   1:L PR[91] R[100]mm/sec CNT100;
   1:  PR[91,1] = PR[90,1] + 29.253;
   1:  PR[91,2] = PR[90,2] + 16.282;
   1:L PR[91] R[100]mm/sec CNT100;
   1:  PR[91,1] = PR[90,1] + 26.405;
   1:  PR[91,2] = PR[90,2] + 17.087;
   1:L PR[91] R[100]mm/sec CNT100;
   1:  PR[91,1] = PR[90,1] + 25.337;
   1:  PR[91,2] = PR[90,2] + 17.312;
   1:L PR[91] R[100]mm/sec CNT100;
   1:  PR[91,1] = PR[90,1] + 24.258;
   1:  PR[91,2] = PR[90,2] + 17.381;
   1:L PR[91] R[100]mm/sec CNT100;
   1:  PR[91,1] = PR[90,1] + 21.299;
   1:  PR[91,2] = PR[90,2] + 17.344;
   1:L PR[91] R[100]mm/sec CNT100;
   1:  PR[91,1] = PR[90,1] + 20.210;
   1:  PR[91,2] = PR[90,2] + 17.257;
   1:L PR[91] R[100]mm/sec CNT100;
   1:  PR[91,1] = PR[90,1] + 19.156;
   1:  PR[91,2] = PR[90,2] + 17.019;
   1:L PR[91] R[100]mm/sec CNT100;
   1:  PR[91,1] = PR[90,1] + 16.330;
   1:  PR[91,2] = PR[90,2] + 16.144;
   1:L PR[91] R[100]mm/sec CNT100;
   1:  PR[91,1] = PR[90,1] + 15.309;
   1:  PR[91,2] = PR[90,2] + 15.752;
   1:L PR[91] R[100]mm/sec CNT100;
   1:  PR[91,1] = PR[90,1] + 14.367;
   1:  PR[91,2] = PR[90,2] + 15.225;
   1:L PR[91] R[100]mm/sec CNT100;
   1:  PR[91,1] = PR[90,1] + 11.906;
   1:  PR[91,2] = PR[90,2] + 13.584;
   1:L PR[91] R[100]mm/sec CNT100;
   1:  PR[91,1] = PR[90,1] + 11.037;
   1:  PR[91,2] = PR[90,2] + 12.919;
   1:L PR[91] R[100]mm/sec CNT100;
   1:  PR[91,1] = PR[90,1] + 10.284;
   1:  PR[91,2] = PR[90,2] + 12.148;
   1:L PR[91] R[100]mm/sec CNT100;
   1:  PR[91,1] = PR[90,1] + 8.389;
   1:  PR[91,2] = PR[90,2] + 9.875;
   1:L PR[91] R[100]mm/sec CNT100;
   1:  PR[91,1] = PR[90,1] + 7.743;
   1:  PR[91,2] = PR[90,2] + 8.991;
   1:L PR[91] R[100]mm/sec CNT100;
   1:  PR[91,1] = PR[90,1] + 7.239;
   1:  PR[91,2] = PR[90,2] + 8.038;
   1:L PR[91] R[100]mm/sec CNT100;
   1:  PR[91,1] = PR[90,1] + 6.070;
   1:  PR[91,2] = PR[90,2] + 5.329;
   1:L PR[91] R[100]mm/sec CNT100;
   1:  PR[91,1] = PR[90,1] + 5.524;
   1:  PR[91,2] = PR[90,2] + 3.781;
   1:L PR[91] R[100]mm/sec CNT100;
   1:  PR[91,1] = PR[90,1] + 4.280;
   1:  PR[91,2] = PR[90,2] + 1.925;
   1:L PR[91] R[100]mm/sec CNT100;
   1:  PR[91,1] = PR[90,1] + 2.077;
   1:  PR[91,2] = PR[90,2] + 1.178;
   1:L PR[91] R[100]mm/sec CNT100;
   1:  PR[91] = PR[90];
   1:  PR[91,1] = PR[90,1] + -2.557;
   1:  PR[91,3] = PR[90,3] + 4.095;
   1:L PR[91] R[100]mm/sec CNT100;
   1:  PR[91,1] = PR[90,1] + -4.760;
   1:  PR[91,2] = PR[90,2] + 1.925;
   1:L PR[91] R[100]mm/sec CNT100;
   1:  PR[91,1] = PR[90,1] + -5.964;
   1:  PR[91,2] = PR[90,2] + 3.722;
   1:L PR[91] R[100]mm/sec CNT100;
   1:  PR[91,1] = PR[90,1] + -6.705;
   1:  PR[91,2] = PR[90,2] + 5.489;
   1:L PR[91] R[100]mm/sec CNT100;
   1:  PR[91,1] = PR[90,1] + -7.396;
   1:  PR[91,2] = PR[90,2] + 7.422;
   1:L PR[91] R[100]mm/sec CNT100;
   1:  PR[91,1] = PR[90,1] + -8.209;
   1:  PR[91,2] = PR[90,2] + 8.958;
   1:L PR[91] R[100]mm/sec CNT100;
   1:  PR[91,1] = PR[90,1] + -9.058;
   1:  PR[91,2] = PR[90,2] + 9.976;
   1:L PR[91] R[100]mm/sec CNT100;
   1:  PR[91,1] = PR[90,1] + -10.276;
   1:  PR[91,2] = PR[90,2] + 11.645;
   1:L PR[91] R[100]mm/sec CNT100;
   1:  PR[91,1] = PR[90,1] + -11.490;
   1:  PR[91,2] = PR[90,2] + 12.888;
   1:L PR[91] R[100]mm/sec CNT100;
   1:  PR[91,1] = PR[90,1] + -12.593;
   1:  PR[91,2] = PR[90,2] + 13.623;
   1:L PR[91] R[100]mm/sec CNT100;
   1:  PR[91,1] = PR[90,1] + -14.234;
   1:  PR[91,2] = PR[90,2] + 14.880;
   1:L PR[91] R[100]mm/sec CNT100;
   1:  PR[91,1] = PR[90,1] + -15.750;
   1:  PR[91,2] = PR[90,2] + 15.727;
   1:L PR[91] R[100]mm/sec CNT100;
   1:  PR[91,1] = PR[90,1] + -17.017;
   1:  PR[91,2] = PR[90,2] + 16.119;
   1:L PR[91] R[100]mm/sec CNT100;
   1:  PR[91,1] = PR[90,1] + -18.947;
   1:  PR[91,2] = PR[90,2] + 16.860;
   1:L PR[91] R[100]mm/sec CNT100;
   1:  PR[91,1] = PR[90,1] + -20.639;
   1:  PR[91,2] = PR[90,2] + 17.244;
   1:L PR[91] R[100]mm/sec CNT100;
   1:  PR[91,1] = PR[90,1] + -21.966;
   1:  PR[91,2] = PR[90,2] + 17.260;
   1:L PR[91] R[100]mm/sec CNT100;
   1:  PR[91,1] = PR[90,1] + -24.028;
   1:  PR[91,2] = PR[90,2] + 17.425;
   1:L PR[91] R[100]mm/sec CNT100;
   1:  PR[91,1] = PR[90,1] + -25.758;
   1:  PR[91,2] = PR[90,2] + 17.314;
   1:L PR[91] R[100]mm/sec CNT100;
   1:  PR[91,1] = PR[90,1] + -27.035;
   1:  PR[91,2] = PR[90,2] + 16.953;
   1:L PR[91] R[100]mm/sec CNT100;
   1:  PR[91,1] = PR[90,1] + -29.061;
   1:  PR[91,2] = PR[90,2] + 16.526;
   1:L PR[91] R[100]mm/sec CNT100;
   1:  PR[91,1] = PR[90,1] + -30.688;
   1:  PR[91,2] = PR[90,2] + 15.930;
   1:L PR[91] R[100]mm/sec CNT100;
   1:  PR[91,1] = PR[90,1] + -31.809;
   1:  PR[91,2] = PR[90,2] + 15.222;
   1:L PR[91] R[100]mm/sec CNT100;
   1:  PR[91,1] = PR[90,1] + -33.632;
   1:  PR[91,2] = PR[90,2] + 14.239;
   1:L PR[91] R[100]mm/sec CNT100;
   1:  PR[91,1] = PR[90,1] + -35.023;
   1:  PR[91,2] = PR[90,2] + 13.207;
   1:L PR[91] R[100]mm/sec CNT100;
   1:  PR[91,1] = PR[90,1] + -35.897;
   1:  PR[91,2] = PR[90,2] + 12.210;
   1:L PR[91] R[100]mm/sec CNT100;
   1:  PR[91,1] = PR[90,1] + -37.368;
   1:  PR[91,2] = PR[90,2] + 10.751;
   1:L PR[91] R[100]mm/sec CNT100;
   1:  PR[91,1] = PR[90,1] + -38.410;
   1:  PR[91,2] = PR[90,2] + 9.368;
   1:L PR[91] R[100]mm/sec CNT100;
   1:  PR[91,1] = PR[90,1] + -38.965;
   1:  PR[91,2] = PR[90,2] + 8.164;
   1:L PR[91] R[100]mm/sec CNT100;
   1:  PR[91,1] = PR[90,1] + -39.963;
   1:  PR[91,2] = PR[90,2] + 6.347;
   1:L PR[91] R[100]mm/sec CNT100;
   1:  PR[91,1] = PR[90,1] + -40.570;
   1:  PR[91,2] = PR[90,2] + 4.727;
   1:L PR[91] R[100]mm/sec CNT100;
   1:  PR[91,1] = PR[90,1] + -40.760;
   1:  PR[91,2] = PR[90,2] + 3.414;
   1:L PR[91] R[100]mm/sec CNT100;
   1:  PR[91,1] = PR[90,1] + -41.203;
   1:  PR[91,2] = PR[90,2] + 1.388;
   1:L PR[91] R[100]mm/sec CNT100;
   1:  PR[91,1] = PR[90,1] + -41.327;
   1:  PR[91,2] = PR[90,2] + -0.336;
   1:L PR[91] R[100]mm/sec CNT100;
   1:  PR[91,1] = PR[90,1] + -41.137;
   1:  PR[91,2] = PR[90,2] + -1.650;
   1:L PR[91] R[100]mm/sec CNT100;
   1:  PR[91,1] = PR[90,1] + -40.988;
   1:  PR[91,2] = PR[90,2] + -3.720;
   1:L PR[91] R[100]mm/sec CNT100;
   1:  PR[91,1] = PR[90,1] + -40.600;
   1:  PR[91,2] = PR[90,2] + -5.494;
   1:L PR[91] R[100]mm/sec CNT100;
   1:  PR[91,1] = PR[90,1] + -39.933;
   1:  PR[91,2] = PR[90,2] + -7.273;
   1:L PR[91] R[100]mm/sec CNT100;
   1:  PR[91,1] = PR[90,1] + -39.377;
   1:  PR[91,2] = PR[90,2] + -8.479;
   1:L PR[91] R[100]mm/sec CNT100;
   1:  PR[91,1] = PR[90,1] + -38.461;
   1:  PR[91,2] = PR[90,2] + -10.147;
   1:L PR[91] R[100]mm/sec CNT100;
   1:  PR[91,1] = PR[90,1] + -37.318;
   1:  PR[91,2] = PR[90,2] + -11.665;
   1:L PR[91] R[100]mm/sec CNT100;
   1:  PR[91,1] = PR[90,1] + -36.443;
   1:  PR[91,2] = PR[90,2] + -12.663;
   1:L PR[91] R[100]mm/sec CNT100;
   1:  PR[91,1] = PR[90,1] + -35.091;
   1:  PR[91,2] = PR[90,2] + -14.005;
   1:L PR[91] R[100]mm/sec CNT100;
   1:  PR[91,1] = PR[90,1] + -33.566;
   1:  PR[91,2] = PR[90,2] + -15.135;
   1:L PR[91] R[100]mm/sec CNT100;
   1:  PR[91,1] = PR[90,1] + -32.443;
   1:  PR[91,2] = PR[90,2] + -15.844;
   1:L PR[91] R[100]mm/sec CNT100;
   1:  PR[91,1] = PR[90,1] + -30.766;
   1:  PR[91,2] = PR[90,2] + -16.749;
   1:L PR[91] R[100]mm/sec CNT100;
   1:  PR[91,1] = PR[90,1] + -28.984;
   1:  PR[91,2] = PR[90,2] + -17.401;
   1:L PR[91] R[100]mm/sec CNT100;
   1:  PR[91,1] = PR[90,1] + -27.706;
   1:  PR[91,2] = PR[90,2] + -17.763;
   1:L PR[91] R[100]mm/sec CNT100;
   1:  PR[91,1] = PR[90,1] + -25.840;
   1:  PR[91,2] = PR[90,2] + -18.156;
   1:L PR[91] R[100]mm/sec CNT100;
   1:  PR[91,1] = PR[90,1] + -23.948;
   1:  PR[91,2] = PR[90,2] + -18.277;
   1:L PR[91] R[100]mm/sec CNT100;
   1:  PR[91,1] = PR[90,1] + -22.620;
   1:  PR[91,2] = PR[90,2] + -18.261;
   1:L PR[91] R[100]mm/sec CNT100;
   1:  PR[91,1] = PR[90,1] + -20.718;
   1:  PR[91,2] = PR[90,2] + -18.109;
   1:L PR[91] R[100]mm/sec CNT100;
   1:  PR[91,1] = PR[90,1] + -18.869;
   1:  PR[91,2] = PR[90,2] + -17.690;
   1:L PR[91] R[100]mm/sec CNT100;
   1:  PR[91,1] = PR[90,1] + -17.602;
   1:  PR[91,2] = PR[90,2] + -17.297;
   1:L PR[91] R[100]mm/sec CNT100;
   1:  PR[91,1] = PR[90,1] + -15.819;
   1:  PR[91,2] = PR[90,2] + -16.613;
   1:L PR[91] R[100]mm/sec CNT100;
   1:  PR[91,1] = PR[90,1] + -14.166;
   1:  PR[91,2] = PR[90,2] + -15.689;
   1:L PR[91] R[100]mm/sec CNT100;
   1:  PR[91,1] = PR[90,1] + -13.062;
   1:  PR[91,2] = PR[90,2] + -14.953;
   1:L PR[91] R[100]mm/sec CNT100;
   1:  PR[91,1] = PR[90,1] + -11.545;
   1:  PR[91,2] = PR[90,2] + -13.792;
   1:L PR[91] R[100]mm/sec CNT100;
   1:  PR[91,1] = PR[90,1] + -10.222;
   1:  PR[91,2] = PR[90,2] + -12.437;
   1:L PR[91] R[100]mm/sec CNT100;
   1:  PR[91,1] = PR[90,1] + -9.372;
   1:  PR[91,2] = PR[90,2] + -11.418;
   1:L PR[91] R[100]mm/sec CNT100;
   1:  PR[91,1] = PR[90,1] + -8.245;
   1:  PR[91,2] = PR[90,2] + -9.874;
   1:L PR[91] R[100]mm/sec CNT100;
   1:  PR[91,1] = PR[90,1] + -7.360;
   1:  PR[91,2] = PR[90,2] + -8.201;
   1:L PR[91] R[100]mm/sec CNT100;
   1:  PR[91,1] = PR[90,1] + -6.836;
   1:  PR[91,2] = PR[90,2] + -6.988;
   1:L PR[91] R[100]mm/sec CNT100;
   1:  PR[91,1] = PR[90,1] + -6.003;
   1:  PR[91,2] = PR[90,2] + -4.628;
   1:L PR[91] R[100]mm/sec CNT100;
   1:  PR[91,1] = PR[90,1] + -4.760;
   1:  PR[91,2] = PR[90,2] + -2.772;
   1:L PR[91] R[100]mm/sec CNT100;
   1:  PR[91,1] = PR[90,1] + -2.557;
   1:  PR[91,2] = PR[90,2] + -2.026;
   1:L PR[91] R[100]mm/sec CNT100;
   1:  PR[91,1] = PR[90,1] + 2.077;
   1:L PR[91] R[100]mm/sec CNT100;
   1:  PR[91,1] = PR[90,1] + 4.280;
   1:  PR[91,2] = PR[90,2] + -2.772;
   1:L PR[91] R[100]mm/sec CNT100;
   1:  PR[91,1] = PR[90,1] + 5.485;
   1:  PR[91,2] = PR[90,2] + -4.570;
   1:L PR[91] R[100]mm/sec CNT100;
   1:  PR[91,1] = PR[90,1] + 6.225;
   1:  PR[91,2] = PR[90,2] + -6.336;
   1:L PR[91] R[100]mm/sec CNT100;
   1:  PR[91,1] = PR[90,1] + 6.916;
   1:  PR[91,2] = PR[90,2] + -8.269;
   1:L PR[91] R[100]mm/sec CNT100;
   1:  PR[91,1] = PR[90,1] + 7.729;
   1:  PR[91,2] = PR[90,2] + -9.805;
   1:L PR[91] R[100]mm/sec CNT100;
   1:  PR[91,1] = PR[90,1] + 8.579;
   1:  PR[91,2] = PR[90,2] + -10.824;
   1:L PR[91] R[100]mm/sec CNT100;
   1:  PR[91,1] = PR[90,1] + 9.796;
   1:  PR[91,2] = PR[90,2] + -12.493;
   1:L PR[91] R[100]mm/sec CNT100;
   1:  PR[91,1] = PR[90,1] + 11.010;
   1:  PR[91,2] = PR[90,2] + -13.735;
   1:L PR[91] R[100]mm/sec CNT100;
   1:  PR[91,1] = PR[90,1] + 12.114;
   1:  PR[91,2] = PR[90,2] + -14.471;
   1:L PR[91] R[100]mm/sec CNT100;
   1:  PR[91,1] = PR[90,1] + 13.755;
   1:  PR[91,2] = PR[90,2] + -15.727;
   1:L PR[91] R[100]mm/sec CNT100;
   1:  PR[91,1] = PR[90,1] + 15.270;
   1:  PR[91,2] = PR[90,2] + -16.574;
   1:L PR[91] R[100]mm/sec CNT100;
   1:  PR[91,1] = PR[90,1] + 16.537;
   1:  PR[91,2] = PR[90,2] + -16.967;
   1:L PR[91] R[100]mm/sec CNT100;
   1:  PR[91,1] = PR[90,1] + 18.467;
   1:  PR[91,2] = PR[90,2] + -17.708;
   1:L PR[91] R[100]mm/sec CNT100;
   1:  PR[91,1] = PR[90,1] + 20.159;
   1:  PR[91,2] = PR[90,2] + -18.091;
   1:L PR[91] R[100]mm/sec CNT100;
   1:  PR[91,1] = PR[90,1] + 21.486;
   1:  PR[91,2] = PR[90,2] + -18.108;
   1:L PR[91] R[100]mm/sec CNT100;
   1:  PR[91,1] = PR[90,1] + 23.549;
   1:  PR[91,2] = PR[90,2] + -18.272;
   1:L PR[91] R[100]mm/sec CNT100;
   1:  PR[91,1] = PR[90,1] + 25.279;
   1:  PR[91,2] = PR[90,2] + -18.161;
   1:L PR[91] R[100]mm/sec CNT100;
   1:  PR[91,1] = PR[90,1] + 26.555;
   1:  PR[91,2] = PR[90,2] + -17.800;
   1:L PR[91] R[100]mm/sec CNT100;
   1:  PR[91,1] = PR[90,1] + 28.581;
   1:  PR[91,2] = PR[90,2] + -17.373;
   1:L PR[91] R[100]mm/sec CNT100;
   1:  PR[91,1] = PR[90,1] + 30.208;
   1:  PR[91,2] = PR[90,2] + -16.778;
   1:L PR[91] R[100]mm/sec CNT100;
   1:  PR[91,1] = PR[90,1] + 31.330;
   1:  PR[91,2] = PR[90,2] + -16.069;
   1:L PR[91] R[100]mm/sec CNT100;
   1:  PR[91,1] = PR[90,1] + 33.152;
   1:  PR[91,2] = PR[90,2] + -15.086;
   1:L PR[91] R[100]mm/sec CNT100;
   1:  PR[91,1] = PR[90,1] + 34.543;
   1:  PR[91,2] = PR[90,2] + -14.055;
   1:L PR[91] R[100]mm/sec CNT100;
   1:  PR[91,1] = PR[90,1] + 35.418;
   1:  PR[91,2] = PR[90,2] + -13.057;
   1:L PR[91] R[100]mm/sec CNT100;
   1:  PR[91,1] = PR[90,1] + 36.888;
   1:  PR[91,2] = PR[90,2] + -11.598;
   1:L PR[91] R[100]mm/sec CNT100;
   1:  PR[91,1] = PR[90,1] + 37.930;
   1:  PR[91,2] = PR[90,2] + -10.215;
   1:L PR[91] R[100]mm/sec CNT100;
   1:  PR[91,1] = PR[90,1] + 38.485;
   1:  PR[91,2] = PR[90,2] + -9.011;
   1:L PR[91] R[100]mm/sec CNT100;
   1:  PR[91,1] = PR[90,1] + 39.483;
   1:  PR[91,2] = PR[90,2] + -7.194;
   1:L PR[91] R[100]mm/sec CNT100;
   1:  PR[91,1] = PR[90,1] + 40.090;
   1:  PR[91,2] = PR[90,2] + -5.574;
   1:L PR[91] R[100]mm/sec CNT100;
   1:  PR[91,1] = PR[90,1] + 40.281;
   1:  PR[91,2] = PR[90,2] + -4.261;
   1:L PR[91] R[100]mm/sec CNT100;
   1:  PR[91,1] = PR[90,1] + 40.724;
   1:  PR[91,2] = PR[90,2] + -2.235;
   1:L PR[91] R[100]mm/sec CNT100;
   1:  PR[91,1] = PR[90,1] + 40.848;
   1:  PR[91,2] = PR[90,2] + -0.511;
   1:L PR[91] R[100]mm/sec CNT100;
   1:  PR[91,1] = PR[90,1] + 40.657;
   1:  PR[91,2] = PR[90,2] + 0.802;
   1:L PR[91] R[100]mm/sec CNT100;
   1:  PR[91,1] = PR[90,1] + 40.509;
   1:  PR[91,2] = PR[90,2] + 2.872;
   1:L PR[91] R[100]mm/sec CNT100;
   1:  PR[91,1] = PR[90,1] + 40.121;
   1:  PR[91,2] = PR[90,2] + 4.646;
   1:L PR[91] R[100]mm/sec CNT100;
   1:  PR[91,1] = PR[90,1] + 39.453;
   1:  PR[91,2] = PR[90,2] + 6.426;
   1:L PR[91] R[100]mm/sec CNT100;
   1:  PR[91,1] = PR[90,1] + 38.898;
   1:  PR[91,2] = PR[90,2] + 7.631;
   1:L PR[91] R[100]mm/sec CNT100;
   1:  PR[91,1] = PR[90,1] + 37.981;
   1:  PR[91,2] = PR[90,2] + 9.300;
   1:L PR[91] R[100]mm/sec CNT100;
   1:  PR[91,1] = PR[90,1] + 36.838;
   1:  PR[91,2] = PR[90,2] + 10.817;
   1:L PR[91] R[100]mm/sec CNT100;
   1:  PR[91,1] = PR[90,1] + 35.963;
   1:  PR[91,2] = PR[90,2] + 11.816;
   1:L PR[91] R[100]mm/sec CNT100;
   1:  PR[91,1] = PR[90,1] + 34.611;
   1:  PR[91,2] = PR[90,2] + 13.157;
   1:L PR[91] R[100]mm/sec CNT100;
   1:  PR[91,1] = PR[90,1] + 33.086;
   1:  PR[91,2] = PR[90,2] + 14.288;
   1:L PR[91] R[100]mm/sec CNT100;
   1:  PR[91,1] = PR[90,1] + 31.964;
   1:  PR[91,2] = PR[90,2] + 14.997;
   1:L PR[91] R[100]mm/sec CNT100;
   1:  PR[91,1] = PR[90,1] + 30.286;
   1:  PR[91,2] = PR[90,2] + 15.902;
   1:L PR[91] R[100]mm/sec CNT100;
   1:  PR[91,1] = PR[90,1] + 28.504;
   1:  PR[91,2] = PR[90,2] + 16.554;
   1:L PR[91] R[100]mm/sec CNT100;
   1:  PR[91,1] = PR[90,1] + 27.227;
   1:  PR[91,2] = PR[90,2] + 16.915;
   1:L PR[91] R[100]mm/sec CNT100;
   1:  PR[91,1] = PR[90,1] + 25.361;
   1:  PR[91,2] = PR[90,2] + 17.308;
   1:L PR[91] R[100]mm/sec CNT100;
   1:  PR[91,1] = PR[90,1] + 23.468;
   1:  PR[91,2] = PR[90,2] + 17.430;
   1:L PR[91] R[100]mm/sec CNT100;
   1:  PR[91,1] = PR[90,1] + 22.140;
   1:  PR[91,2] = PR[90,2] + 17.413;
   1:L PR[91] R[100]mm/sec CNT100;
   1:  PR[91,1] = PR[90,1] + 20.238;
   1:  PR[91,2] = PR[90,2] + 17.262;
   1:L PR[91] R[100]mm/sec CNT100;
   1:  PR[91,1] = PR[90,1] + 18.390;
   1:  PR[91,2] = PR[90,2] + 16.843;
   1:L PR[91] R[100]mm/sec CNT100;
   1:  PR[91,1] = PR[90,1] + 17.122;
   1:  PR[91,2] = PR[90,2] + 16.450;
   1:L PR[91] R[100]mm/sec CNT100;
   1:  PR[91,1] = PR[90,1] + 15.340;
   1:  PR[91,2] = PR[90,2] + 15.766;
   1:L PR[91] R[100]mm/sec CNT100;
   1:  PR[91,1] = PR[90,1] + 13.686;
   1:  PR[91,2] = PR[90,2] + 14.841;
   1:L PR[91] R[100]mm/sec CNT100;
   1:  PR[91,1] = PR[90,1] + 12.582;
   1:  PR[91,2] = PR[90,2] + 14.105;
   1:L PR[91] R[100]mm/sec CNT100;
   1:  PR[91,1] = PR[90,1] + 11.066;
   1:  PR[91,2] = PR[90,2] + 12.944;
   1:L PR[91] R[100]mm/sec CNT100;
   1:  PR[91,1] = PR[90,1] + 9.742;
   1:  PR[91,2] = PR[90,2] + 11.590;
   1:L PR[91] R[100]mm/sec CNT100;
   1:  PR[91,1] = PR[90,1] + 8.892;
   1:  PR[91,2] = PR[90,2] + 10.570;
   1:L PR[91] R[100]mm/sec CNT100;
   1:  PR[91,1] = PR[90,1] + 7.766;
   1:  PR[91,2] = PR[90,2] + 9.027;
   1:L PR[91] R[100]mm/sec CNT100;
   1:  PR[91,1] = PR[90,1] + 6.880;
   1:  PR[91,2] = PR[90,2] + 7.354;
   1:L PR[91] R[100]mm/sec CNT100;
   1:  PR[91,1] = PR[90,1] + 6.357;
   1:  PR[91,2] = PR[90,2] + 6.141;
   1:L PR[91] R[100]mm/sec CNT100;
   1:  PR[91,1] = PR[90,1] + 5.524;
   1:  PR[91,2] = PR[90,2] + 3.781;
   1:L PR[91] R[100]mm/sec CNT100;
   1:  PR[91,1] = PR[90,1] + 4.280;
   1:  PR[91,2] = PR[90,2] + 1.925;
   1:L PR[91] R[100]mm/sec CNT100;
   1:  PR[91,1] = PR[90,1] + 2.077;
   1:  PR[91,2] = PR[90,2] + 1.178;
   1:L PR[91] R[100]mm/sec CNT100;
   1:  PR[91] = PR[90];
   1:  PR[91,1] = PR[90,1] + -2.588;
   1:  PR[91,2] = PR[90,2] + 1.338;
   1:  PR[91,3] = PR[90,3] + 5.395;
   1:L PR[91] R[100]mm/sec CNT100;
   1:  PR[91,1] = PR[90,1] + -3.756;
   1:  PR[91,2] = PR[90,2] + 1.733;
   1:L PR[91] R[100]mm/sec CNT100;
   1:  PR[91,1] = PR[90,1] + -4.826;
   1:  PR[91,2] = PR[90,2] + 2.147;
   1:L PR[91] R[100]mm/sec CNT100;
   1:  PR[91,1] = PR[90,1] + -6.051;
   1:  PR[91,2] = PR[90,2] + 3.962;
   1:L PR[91] R[100]mm/sec CNT100;
   1:  PR[91,1] = PR[90,1] + -7.046;
   1:  PR[91,2] = PR[90,2] + 6.761;
   1:L PR[91] R[100]mm/sec CNT100;
   1:  PR[91,1] = PR[90,1] + -8.266;
   1:  PR[91,2] = PR[90,2] + 9.072;
   1:L PR[91] R[100]mm/sec CNT100;
   1:  PR[91,1] = PR[90,1] + -9.737;
   1:  PR[91,2] = PR[90,2] + 11.088;
   1:L PR[91] R[100]mm/sec CNT100;
   1:  PR[91,1] = PR[90,1] + -11.556;
   1:  PR[91,2] = PR[90,2] + 12.960;
   1:L PR[91] R[100]mm/sec CNT100;
   1:  PR[91,1] = PR[90,1] + -13.623;
   1:  PR[91,2] = PR[90,2] + 14.542;
   1:L PR[91] R[100]mm/sec CNT100;
   1:  PR[91,1] = PR[90,1] + -15.809;
   1:  PR[91,2] = PR[90,2] + 15.764;
   1:L PR[91] R[100]mm/sec CNT100;
   1:  PR[91,1] = PR[90,1] + -18.238;
   1:  PR[91,2] = PR[90,2] + 16.700;
   1:L PR[91] R[100]mm/sec CNT100;
   1:  PR[91,1] = PR[90,1] + -20.774;
   1:  PR[91,2] = PR[90,2] + 17.271;
   1:L PR[91] R[100]mm/sec CNT100;
   1:  PR[91,1] = PR[90,1] + -23.277;
   1:  PR[91,2] = PR[90,2] + 17.470;
   1:L PR[91] R[100]mm/sec CNT100;
   1:  PR[91,1] = PR[90,1] + -25.872;
   1:  PR[91,2] = PR[90,2] + 17.304;
   1:L PR[91] R[100]mm/sec CNT100;
   1:  PR[91,1] = PR[90,1] + -28.332;
   1:  PR[91,2] = PR[90,2] + 16.786;
   1:L PR[91] R[100]mm/sec CNT100;
   1:  PR[91,1] = PR[90,1] + -30.774;
   1:  PR[91,2] = PR[90,2] + 15.897;
   1:L PR[91] R[100]mm/sec CNT100;
   1:  PR[91,1] = PR[90,1] + -33.056;
   1:  PR[91,2] = PR[90,2] + 14.664;
   1:L PR[91] R[100]mm/sec CNT100;
   1:  PR[91,1] = PR[90,1] + -35.079;
   1:  PR[91,2] = PR[90,2] + 13.164;
   1:L PR[91] R[100]mm/sec CNT100;
   1:  PR[91,1] = PR[90,1] + -36.921;
   1:  PR[91,2] = PR[90,2] + 11.338;
   1:L PR[91] R[100]mm/sec CNT100;
   1:  PR[91,1] = PR[90,1] + -38.478;
   1:  PR[91,2] = PR[90,2] + 9.264;
   1:L PR[91] R[100]mm/sec CNT100;
   1:  PR[91,1] = PR[90,1] + -39.692;
   1:  PR[91,2] = PR[90,2] + 7.054;
   1:L PR[91] R[100]mm/sec CNT100;
   1:  PR[91,1] = PR[90,1] + -40.602;
   1:  PR[91,2] = PR[90,2] + 4.626;
   1:L PR[91] R[100]mm/sec CNT100;
   1:  PR[91,1] = PR[90,1] + -41.141;
   1:  PR[91,2] = PR[90,2] + 2.162;
   1:L PR[91] R[100]mm/sec CNT100;
   1:  PR[91,1] = PR[90,1] + -41.330;
   1:  PR[91,2] = PR[90,2] + -0.424;
   1:L PR[91] R[100]mm/sec CNT100;
   1:  PR[91,1] = PR[90,1] + -41.141;
   1:  PR[91,2] = PR[90,2] + -3.009;
   1:L PR[91] R[100]mm/sec CNT100;
   1:  PR[91,1] = PR[90,1] + -40.602;
   1:  PR[91,2] = PR[90,2] + -5.473;
   1:L PR[91] R[100]mm/sec CNT100;
   1:  PR[91,1] = PR[90,1] + -39.692;
   1:  PR[91,2] = PR[90,2] + -7.902;
   1:L PR[91] R[100]mm/sec CNT100;
   1:  PR[91,1] = PR[90,1] + -38.478;
   1:  PR[91,2] = PR[90,2] + -10.112;
   1:L PR[91] R[100]mm/sec CNT100;
   1:  PR[91,1] = PR[90,1] + -36.921;
   1:  PR[91,2] = PR[90,2] + -12.186;
   1:L PR[91] R[100]mm/sec CNT100;
   1:  PR[91,1] = PR[90,1] + -35.132;
   1:  PR[91,2] = PR[90,2] + -13.961;
   1:L PR[91] R[100]mm/sec CNT100;
   1:  PR[91,1] = PR[90,1] + -33.053;
   1:  PR[91,2] = PR[90,2] + -15.513;
   1:L PR[91] R[100]mm/sec CNT100;
   1:  PR[91,1] = PR[90,1] + -30.774;
   1:  PR[91,2] = PR[90,2] + -16.744;
   1:L PR[91] R[100]mm/sec CNT100;
   1:  PR[91,1] = PR[90,1] + -28.332;
   1:  PR[91,2] = PR[90,2] + -17.633;
   1:L PR[91] R[100]mm/sec CNT100;
   1:  PR[91,1] = PR[90,1] + -25.872;
   1:  PR[91,2] = PR[90,2] + -18.151;
   1:L PR[91] R[100]mm/sec CNT100;
   1:  PR[91,1] = PR[90,1] + -23.277;
   1:  PR[91,2] = PR[90,2] + -18.317;
   1:L PR[91] R[100]mm/sec CNT100;
   1:  PR[91,1] = PR[90,1] + -20.774;
   1:  PR[91,2] = PR[90,2] + -18.118;
   1:L PR[91] R[100]mm/sec CNT100;
   1:  PR[91,1] = PR[90,1] + -18.238;
   1:  PR[91,2] = PR[90,2] + -17.547;
   1:L PR[91] R[100]mm/sec CNT100;
   1:  PR[91,1] = PR[90,1] + -15.809;
   1:  PR[91,2] = PR[90,2] + -16.611;
   1:L PR[91] R[100]mm/sec CNT100;
   1:  PR[91,1] = PR[90,1] + -13.623;
   1:  PR[91,2] = PR[90,2] + -15.389;
   1:L PR[91] R[100]mm/sec CNT100;
   1:  PR[91,1] = PR[90,1] + -11.553;
   1:  PR[91,2] = PR[90,2] + -13.805;
   1:L PR[91] R[100]mm/sec CNT100;
   1:  PR[91,1] = PR[90,1] + -9.805;
   1:  PR[91,2] = PR[90,2] + -12.017;
   1:L PR[91] R[100]mm/sec CNT100;
   1:  PR[91,1] = PR[90,1] + -8.264;
   1:  PR[91,2] = PR[90,2] + -9.915;
   1:L PR[91] R[100]mm/sec CNT100;
   1:  PR[91,1] = PR[90,1] + -7.047;
   1:  PR[91,2] = PR[90,2] + -7.613;
   1:L PR[91] R[100]mm/sec CNT100;
   1:  PR[91,1] = PR[90,1] + -6.052;
   1:  PR[91,2] = PR[90,2] + -4.809;
   1:L PR[91] R[100]mm/sec CNT100;
   1:  PR[91,1] = PR[90,1] + -4.826;
   1:  PR[91,2] = PR[90,2] + -2.994;
   1:L PR[91] R[100]mm/sec CNT100;
   1:  PR[91,1] = PR[90,1] + -3.700;
   1:  PR[91,2] = PR[90,2] + -2.559;
   1:L PR[91] R[100]mm/sec CNT100;
   1:  PR[91,1] = PR[90,1] + -2.587;
   1:  PR[91,2] = PR[90,2] + -2.180;
   1:L PR[91] R[100]mm/sec CNT100;
   1:  PR[91,1] = PR[90,1] + 2.109;
   1:  PR[91,2] = PR[90,2] + -2.185;
   1:L PR[91] R[100]mm/sec CNT100;
   1:  PR[91,1] = PR[90,1] + 3.276;
   1:  PR[91,2] = PR[90,2] + -2.580;
   1:L PR[91] R[100]mm/sec CNT100;
   1:  PR[91,1] = PR[90,1] + 4.346;
   1:  PR[91,2] = PR[90,2] + -2.995;
   1:L PR[91] R[100]mm/sec CNT100;
   1:  PR[91,1] = PR[90,1] + 5.572;
   1:  PR[91,2] = PR[90,2] + -4.809;
   1:L PR[91] R[100]mm/sec CNT100;
   1:  PR[91,1] = PR[90,1] + 6.566;
   1:  PR[91,2] = PR[90,2] + -7.607;
   1:L PR[91] R[100]mm/sec CNT100;
   1:  PR[91,1] = PR[90,1] + 7.786;
   1:  PR[91,2] = PR[90,2] + -9.919;
   1:L PR[91] R[100]mm/sec CNT100;
   1:  PR[91,1] = PR[90,1] + 9.257;
   1:  PR[91,2] = PR[90,2] + -11.935;
   1:L PR[91] R[100]mm/sec CNT100;
   1:  PR[91,1] = PR[90,1] + 11.076;
   1:  PR[91,2] = PR[90,2] + -13.807;
   1:L PR[91] R[100]mm/sec CNT100;
   1:  PR[91,1] = PR[90,1] + 13.144;
   1:  PR[91,2] = PR[90,2] + -15.389;
   1:L PR[91] R[100]mm/sec CNT100;
   1:  PR[91,1] = PR[90,1] + 15.329;
   1:  PR[91,2] = PR[90,2] + -16.611;
   1:L PR[91] R[100]mm/sec CNT100;
   1:  PR[91,1] = PR[90,1] + 17.759;
   1:  PR[91,2] = PR[90,2] + -17.547;
   1:L PR[91] R[100]mm/sec CNT100;
   1:  PR[91,1] = PR[90,1] + 20.295;
   1:  PR[91,2] = PR[90,2] + -18.118;
   1:L PR[91] R[100]mm/sec CNT100;
   1:  PR[91,1] = PR[90,1] + 22.797;
   1:  PR[91,2] = PR[90,2] + -18.317;
   1:L PR[91] R[100]mm/sec CNT100;
   1:  PR[91,1] = PR[90,1] + 25.393;
   1:  PR[91,2] = PR[90,2] + -18.151;
   1:L PR[91] R[100]mm/sec CNT100;
   1:  PR[91,1] = PR[90,1] + 27.852;
   1:  PR[91,2] = PR[90,2] + -17.633;
   1:L PR[91] R[100]mm/sec CNT100;
   1:  PR[91,1] = PR[90,1] + 30.294;
   1:  PR[91,2] = PR[90,2] + -16.744;
   1:L PR[91] R[100]mm/sec CNT100;
   1:  PR[91,1] = PR[90,1] + 32.576;
   1:  PR[91,2] = PR[90,2] + -15.511;
   1:L PR[91] R[100]mm/sec CNT100;
   1:  PR[91,1] = PR[90,1] + 34.599;
   1:  PR[91,2] = PR[90,2] + -14.011;
   1:L PR[91] R[100]mm/sec CNT100;
   1:  PR[91,1] = PR[90,1] + 36.442;
   1:  PR[91,2] = PR[90,2] + -12.185;
   1:L PR[91] R[100]mm/sec CNT100;
   1:  PR[91,1] = PR[90,1] + 37.999;
   1:  PR[91,2] = PR[90,2] + -10.112;
   1:L PR[91] R[100]mm/sec CNT100;
   1:  PR[91,1] = PR[90,1] + 39.213;
   1:  PR[91,2] = PR[90,2] + -7.902;
   1:L PR[91] R[100]mm/sec CNT100;
   1:  PR[91,1] = PR[90,1] + 40.123;
   1:  PR[91,2] = PR[90,2] + -5.473;
   1:L PR[91] R[100]mm/sec CNT100;
   1:  PR[91,1] = PR[90,1] + 40.661;
   1:  PR[91,2] = PR[90,2] + -3.009;
   1:L PR[91] R[100]mm/sec CNT100;
   1:  PR[91,1] = PR[90,1] + 40.850;
   1:  PR[91,2] = PR[90,2] + -0.424;
   1:L PR[91] R[100]mm/sec CNT100;
   1:  PR[91,1] = PR[90,1] + 40.661;
   1:  PR[91,2] = PR[90,2] + 2.162;
   1:L PR[91] R[100]mm/sec CNT100;
   1:  PR[91,1] = PR[90,1] + 40.123;
   1:  PR[91,2] = PR[90,2] + 4.626;
   1:L PR[91] R[100]mm/sec CNT100;
   1:  PR[91,1] = PR[90,1] + 39.213;
   1:  PR[91,2] = PR[90,2] + 7.054;
   1:L PR[91] R[100]mm/sec CNT100;
   1:  PR[91,1] = PR[90,1] + 37.999;
   1:  PR[91,2] = PR[90,2] + 9.264;
   1:L PR[91] R[100]mm/sec CNT100;
   1:  PR[91,1] = PR[90,1] + 36.442;
   1:  PR[91,2] = PR[90,2] + 11.338;
   1:L PR[91] R[100]mm/sec CNT100;
   1:  PR[91,1] = PR[90,1] + 34.599;
   1:  PR[91,2] = PR[90,2] + 13.164;
   1:L PR[91] R[100]mm/sec CNT100;
   1:  PR[91,1] = PR[90,1] + 32.576;
   1:  PR[91,2] = PR[90,2] + 14.664;
   1:L PR[91] R[100]mm/sec CNT100;
   1:  PR[91,1] = PR[90,1] + 30.294;
   1:  PR[91,2] = PR[90,2] + 15.897;
   1:L PR[91] R[100]mm/sec CNT100;
   1:  PR[91,1] = PR[90,1] + 27.852;
   1:  PR[91,2] = PR[90,2] + 16.786;
   1:L PR[91] R[100]mm/sec CNT100;
   1:  PR[91,1] = PR[90,1] + 25.392;
   1:  PR[91,2] = PR[90,2] + 17.304;
   1:L PR[91] R[100]mm/sec CNT100;
   1:  PR[91,1] = PR[90,1] + 22.801;
   1:  PR[91,2] = PR[90,2] + 17.470;
   1:L PR[91] R[100]mm/sec CNT100;
   1:  PR[91,1] = PR[90,1] + 20.206;
   1:  PR[91,2] = PR[90,2] + 17.255;
   1:L PR[91] R[100]mm/sec CNT100;
   1:  PR[91,1] = PR[90,1] + 17.759;
   1:  PR[91,2] = PR[90,2] + 16.700;
   1:L PR[91] R[100]mm/sec CNT100;
   1:  PR[91,1] = PR[90,1] + 15.352;
   1:  PR[91,2] = PR[90,2] + 15.777;
   1:L PR[91] R[100]mm/sec CNT100;
   1:  PR[91,1] = PR[90,1] + 13.144;
   1:  PR[91,2] = PR[90,2] + 14.542;
   1:L PR[91] R[100]mm/sec CNT100;
   1:  PR[91,1] = PR[90,1] + 11.076;
   1:  PR[91,2] = PR[90,2] + 12.960;
   1:L PR[91] R[100]mm/sec CNT100;
   1:  PR[91,1] = PR[90,1] + 9.257;
   1:  PR[91,2] = PR[90,2] + 11.088;
   1:L PR[91] R[100]mm/sec CNT100;
   1:  PR[91,1] = PR[90,1] + 7.785;
   1:  PR[91,2] = PR[90,2] + 9.070;
   1:L PR[91] R[100]mm/sec CNT100;
   1:  PR[91,1] = PR[90,1] + 6.572;
   1:  PR[91,2] = PR[90,2] + 6.779;
   1:L PR[91] R[100]mm/sec CNT100;
   1:  PR[91,1] = PR[90,1] + 5.572;
   1:  PR[91,2] = PR[90,2] + 3.962;
   1:L PR[91] R[100]mm/sec CNT100;
   1:  PR[91,1] = PR[90,1] + 4.346;
   1:  PR[91,2] = PR[90,2] + 2.147;
   1:L PR[91] R[100]mm/sec CNT100;
   1:  PR[91,1] = PR[90,1] + 3.223;
   1:  PR[91,2] = PR[90,2] + 1.713;
   1:L PR[91] R[100]mm/sec CNT100;
   1:  PR[91,1] = PR[90,1] + 2.107;
   1:  PR[91,2] = PR[90,2] + 1.333;
   1:L PR[91] R[100]mm/sec CNT100;
   1:  PR[91] = PR[90];
   1:  PR[91,1] = PR[90,1] + -2.680;
   1:  PR[91,2] = PR[90,2] + 1.767;
   1:  PR[91,3] = PR[90,3] + 6.695;
   1:L PR[91] R[100]mm/sec CNT100;
   1:  PR[91,1] = PR[90,1] + -4.678;
   1:  PR[91,2] = PR[90,2] + 2.508;
   1:L PR[91] R[100]mm/sec CNT100;
   1:  PR[91,1] = PR[90,1] + -5.343;
   1:  PR[91,2] = PR[90,2] + 3.233;
   1:L PR[91] R[100]mm/sec CNT100;
   1:  PR[91,1] = PR[90,1] + -6.128;
   1:  PR[91,2] = PR[90,2] + 4.451;
   1:L PR[91] R[100]mm/sec CNT100;
   1:  PR[91,1] = PR[90,1] + -6.781;
   1:  PR[91,2] = PR[90,2] + 6.328;
   1:L PR[91] R[100]mm/sec CNT100;
   1:  PR[91,1] = PR[90,1] + -7.586;
   1:  PR[91,2] = PR[90,2] + 7.849;
   1:L PR[91] R[100]mm/sec CNT100;
   1:  PR[91,1] = PR[90,1] + -8.268;
   1:  PR[91,2] = PR[90,2] + 9.223;
   1:L PR[91] R[100]mm/sec CNT100;
   1:  PR[91,1] = PR[90,1] + -9.255;
   1:  PR[91,2] = PR[90,2] + 10.575;
   1:L PR[91] R[100]mm/sec CNT100;
   1:  PR[91,1] = PR[90,1] + -10.116;
   1:  PR[91,2] = PR[90,2] + 11.601;
   1:L PR[91] R[100]mm/sec CNT100;
   1:  PR[91,1] = PR[90,1] + -11.333;
   1:  PR[91,2] = PR[90,2] + 12.846;
   1:L PR[91] R[100]mm/sec CNT100;
   1:  PR[91,1] = PR[90,1] + -12.774;
   1:  PR[91,2] = PR[90,2] + 13.949;
   1:L PR[91] R[100]mm/sec CNT100;
   1:  PR[91,1] = PR[90,1] + -13.804;
   1:  PR[91,2] = PR[90,2] + 14.714;
   1:L PR[91] R[100]mm/sec CNT100;
   1:  PR[91,1] = PR[90,1] + -15.310;
   1:  PR[91,2] = PR[90,2] + 15.556;
   1:L PR[91] R[100]mm/sec CNT100;
   1:  PR[91,1] = PR[90,1] + -17.109;
   1:  PR[91,2] = PR[90,2] + 16.247;
   1:L PR[91] R[100]mm/sec CNT100;
   1:  PR[91,1] = PR[90,1] + -18.232;
   1:  PR[91,2] = PR[90,2] + 16.729;
   1:L PR[91] R[100]mm/sec CNT100;
   1:  PR[91,1] = PR[90,1] + -20.012;
   1:  PR[91,2] = PR[90,2] + 17.132;
   1:L PR[91] R[100]mm/sec CNT100;
   1:  PR[91,1] = PR[90,1] + -21.107;
   1:  PR[91,2] = PR[90,2] + 17.325;
   1:L PR[91] R[100]mm/sec CNT100;
   1:  PR[91,1] = PR[90,1] + -22.967;
   1:  PR[91,2] = PR[90,2] + 17.473;
   1:L PR[91] R[100]mm/sec CNT100;
   1:  PR[91,1] = PR[90,1] + -25.993;
   1:  PR[91,2] = PR[90,2] + 17.286;
   1:L PR[91] R[100]mm/sec CNT100;
   1:  PR[91,1] = PR[90,1] + -27.871;
   1:  PR[91,2] = PR[90,2] + 16.890;
   1:L PR[91] R[100]mm/sec CNT100;
   1:  PR[91,1] = PR[90,1] + -28.793;
   1:  PR[91,2] = PR[90,2] + 16.615;
   1:L PR[91] R[100]mm/sec CNT100;
   1:  PR[91,1] = PR[90,1] + -30.656;
   1:  PR[91,2] = PR[90,2] + 15.933;
   1:L PR[91] R[100]mm/sec CNT100;
   1:  PR[91,1] = PR[90,1] + -32.437;
   1:  PR[91,2] = PR[90,2] + 14.973;
   1:L PR[91] R[100]mm/sec CNT100;
   1:  PR[91,1] = PR[90,1] + -33.234;
   1:  PR[91,2] = PR[90,2] + 14.514;
   1:L PR[91] R[100]mm/sec CNT100;
   1:  PR[91,1] = PR[90,1] + -34.799;
   1:  PR[91,2] = PR[90,2] + 13.354;
   1:L PR[91] R[100]mm/sec CNT100;
   1:  PR[91,1] = PR[90,1] + -36.303;
   1:  PR[91,2] = PR[90,2] + 11.862;
   1:L PR[91] R[100]mm/sec CNT100;
   1:  PR[91,1] = PR[90,1] + -36.945;
   1:  PR[91,2] = PR[90,2] + 11.257;
   1:L PR[91] R[100]mm/sec CNT100;
   1:  PR[91,1] = PR[90,1] + -38.150;
   1:  PR[91,2] = PR[90,2] + 9.658;
   1:L PR[91] R[100]mm/sec CNT100;
   1:  PR[91,1] = PR[90,1] + -38.610;
   1:  PR[91,2] = PR[90,2] + 8.960;
   1:L PR[91] R[100]mm/sec CNT100;
   1:  PR[91,1] = PR[90,1] + -39.586;
   1:  PR[91,2] = PR[90,2] + 7.183;
   1:L PR[91] R[100]mm/sec CNT100;
   1:  PR[91,1] = PR[90,1] + -40.611;
   1:  PR[91,2] = PR[90,2] + 4.428;
   1:L PR[91] R[100]mm/sec CNT100;
   1:  PR[91,1] = PR[90,1] + -41.031;
   1:  PR[91,2] = PR[90,2] + 2.506;
   1:L PR[91] R[100]mm/sec CNT100;
   1:  PR[91,1] = PR[90,1] + -41.188;
   1:  PR[91,2] = PR[90,2] + 0.322;
   1:L PR[91] R[100]mm/sec CNT100;
   1:  PR[91,1] = PR[90,1] + -41.281;
   1:  PR[91,2] = PR[90,2] + -0.477;
   1:L PR[91] R[100]mm/sec CNT100;
   1:  PR[91,1] = PR[90,1] + -41.135;
   1:  PR[91,2] = PR[90,2] + -2.510;
   1:L PR[91] R[100]mm/sec CNT100;
   1:  PR[91,1] = PR[90,1] + -41.043;
   1:  PR[91,2] = PR[90,2] + -3.301;
   1:L PR[91] R[100]mm/sec CNT100;
   1:  PR[91,1] = PR[90,1] + -40.611;
   1:  PR[91,2] = PR[90,2] + -5.275;
   1:L PR[91] R[100]mm/sec CNT100;
   1:  PR[91,1] = PR[90,1] + -39.585;
   1:  PR[91,2] = PR[90,2] + -8.031;
   1:L PR[91] R[100]mm/sec CNT100;
   1:  PR[91,1] = PR[90,1] + -38.610;
   1:  PR[91,2] = PR[90,2] + -9.807;
   1:L PR[91] R[100]mm/sec CNT100;
   1:  PR[91,1] = PR[90,1] + -38.150;
   1:  PR[91,2] = PR[90,2] + -10.505;
   1:L PR[91] R[100]mm/sec CNT100;
   1:  PR[91,1] = PR[90,1] + -36.925;
   1:  PR[91,2] = PR[90,2] + -12.130;
   1:L PR[91] R[100]mm/sec CNT100;
   1:  PR[91,1] = PR[90,1] + -35.451;
   1:  PR[91,2] = PR[90,2] + -13.594;
   1:L PR[91] R[100]mm/sec CNT100;
   1:  PR[91,1] = PR[90,1] + -34.825;
   1:  PR[91,2] = PR[90,2] + -14.182;
   1:L PR[91] R[100]mm/sec CNT100;
   1:  PR[91,1] = PR[90,1] + -33.261;
   1:  PR[91,2] = PR[90,2] + -15.342;
   1:L PR[91] R[100]mm/sec CNT100;
   1:  PR[91,1] = PR[90,1] + -31.394;
   1:  PR[91,2] = PR[90,2] + -16.349;
   1:L PR[91] R[100]mm/sec CNT100;
   1:  PR[91,1] = PR[90,1] + -30.623;
   1:  PR[91,2] = PR[90,2] + -16.793;
   1:L PR[91] R[100]mm/sec CNT100;
   1:  PR[91,1] = PR[90,1] + -28.793;
   1:  PR[91,2] = PR[90,2] + -17.463;
   1:L PR[91] R[100]mm/sec CNT100;
   1:  PR[91,1] = PR[90,1] + -27.870;
   1:  PR[91,2] = PR[90,2] + -17.738;
   1:L PR[91] R[100]mm/sec CNT100;
   1:  PR[91,1] = PR[90,1] + -25.992;
   1:  PR[91,2] = PR[90,2] + -18.133;
   1:L PR[91] R[100]mm/sec CNT100;
   1:  PR[91,1] = PR[90,1] + -22.966;
   1:  PR[91,2] = PR[90,2] + -18.321;
   1:L PR[91] R[100]mm/sec CNT100;
   1:  PR[91,1] = PR[90,1] + -21.106;
   1:  PR[91,2] = PR[90,2] + -18.173;
   1:L PR[91] R[100]mm/sec CNT100;
   1:  PR[91,1] = PR[90,1] + -20.011;
   1:  PR[91,2] = PR[90,2] + -17.979;
   1:L PR[91] R[100]mm/sec CNT100;
   1:  PR[91,1] = PR[90,1] + -18.185;
   1:  PR[91,2] = PR[90,2] + -17.565;
   1:L PR[91] R[100]mm/sec CNT100;
   1:  PR[91,1] = PR[90,1] + -16.428;
   1:  PR[91,2] = PR[90,2] + -16.891;
   1:L PR[91] R[100]mm/sec CNT100;
   1:  PR[91,1] = PR[90,1] + -15.351;
   1:  PR[91,2] = PR[90,2] + -16.426;
   1:L PR[91] R[100]mm/sec CNT100;
   1:  PR[91,1] = PR[90,1] + -13.818;
   1:  PR[91,2] = PR[90,2] + -15.569;
   1:L PR[91] R[100]mm/sec CNT100;
   1:  PR[91,1] = PR[90,1] + -12.310;
   1:  PR[91,2] = PR[90,2] + -14.415;
   1:L PR[91] R[100]mm/sec CNT100;
   1:  PR[91,1] = PR[90,1] + -11.319;
   1:  PR[91,2] = PR[90,2] + -13.679;
   1:L PR[91] R[100]mm/sec CNT100;
   1:  PR[91,1] = PR[90,1] + -10.115;
   1:  PR[91,2] = PR[90,2] + -12.447;
   1:L PR[91] R[100]mm/sec CNT100;
   1:  PR[91,1] = PR[90,1] + -9.254;
   1:  PR[91,2] = PR[90,2] + -11.421;
   1:L PR[91] R[100]mm/sec CNT100;
   1:  PR[91,1] = PR[90,1] + -8.248;
   1:  PR[91,2] = PR[90,2] + -10.042;
   1:L PR[91] R[100]mm/sec CNT100;
   1:  PR[91,1] = PR[90,1] + -7.422;
   1:  PR[91,2] = PR[90,2] + -8.481;
   1:L PR[91] R[100]mm/sec CNT100;
   1:  PR[91,1] = PR[90,1] + -6.805;
   1:  PR[91,2] = PR[90,2] + -7.264;
   1:L PR[91] R[100]mm/sec CNT100;
   1:  PR[91,1] = PR[90,1] + -6.652;
   1:  PR[91,2] = PR[90,2] + -6.837;
   1:L PR[91] R[100]mm/sec CNT100;
   1:  PR[91,1] = PR[90,1] + -7.538;
   1:  PR[91,2] = PR[90,2] + -5.744;
   1:L PR[91] R[100]mm/sec CNT100;
   1:  PR[91,1] = PR[90,1] + -5.593;
   1:  PR[91,2] = PR[90,2] + -4.549;
   1:L PR[91] R[100]mm/sec CNT100;
   1:  PR[91,1] = PR[90,1] + -4.910;
   1:  PR[91,2] = PR[90,2] + -3.440;
   1:L PR[91] R[100]mm/sec CNT100;
   1:  PR[91,1] = PR[90,1] + -2.678;
   1:  PR[91,2] = PR[90,2] + -2.614;
   1:L PR[91] R[100]mm/sec CNT100;
   1:  PR[91,1] = PR[90,1] + 2.203;
   1:L PR[91] R[100]mm/sec CNT100;
   1:  PR[91,1] = PR[90,1] + 4.201;
   1:  PR[91,2] = PR[90,2] + -3.356;
   1:L PR[91] R[100]mm/sec CNT100;
   1:  PR[91,1] = PR[90,1] + 4.865;
   1:  PR[91,2] = PR[90,2] + -4.084;
   1:L PR[91] R[100]mm/sec CNT100;
   1:  PR[91,1] = PR[90,1] + 5.648;
   1:  PR[91,2] = PR[90,2] + -5.298;
   1:L PR[91] R[100]mm/sec CNT100;
   1:  PR[91,1] = PR[90,1] + 6.298;
   1:  PR[91,2] = PR[90,2] + -7.164;
   1:L PR[91] R[100]mm/sec CNT100;
   1:  PR[91,1] = PR[90,1] + 7.099;
   1:  PR[91,2] = PR[90,2] + -8.677;
   1:L PR[91] R[100]mm/sec CNT100;
   1:  PR[91,1] = PR[90,1] + 7.788;
   1:  PR[91,2] = PR[90,2] + -10.069;
   1:L PR[91] R[100]mm/sec CNT100;
   1:  PR[91,1] = PR[90,1] + 8.775;
   1:  PR[91,2] = PR[90,2] + -11.421;
   1:L PR[91] R[100]mm/sec CNT100;
   1:  PR[91,1] = PR[90,1] + 9.636;
   1:  PR[91,2] = PR[90,2] + -12.448;
   1:L PR[91] R[100]mm/sec CNT100;
   1:  PR[91,1] = PR[90,1] + 10.853;
   1:  PR[91,2] = PR[90,2] + -13.693;
   1:L PR[91] R[100]mm/sec CNT100;
   1:  PR[91,1] = PR[90,1] + 12.293;
   1:  PR[91,2] = PR[90,2] + -14.796;
   1:L PR[91] R[100]mm/sec CNT100;
   1:  PR[91,1] = PR[90,1] + 13.323;
   1:  PR[91,2] = PR[90,2] + -15.561;
   1:L PR[91] R[100]mm/sec CNT100;
   1:  PR[91,1] = PR[90,1] + 14.829;
   1:  PR[91,2] = PR[90,2] + -16.403;
   1:L PR[91] R[100]mm/sec CNT100;
   1:  PR[91,1] = PR[90,1] + 16.629;
   1:  PR[91,2] = PR[90,2] + -17.094;
   1:L PR[91] R[100]mm/sec CNT100;
   1:  PR[91,1] = PR[90,1] + 17.752;
   1:  PR[91,2] = PR[90,2] + -17.576;
   1:L PR[91] R[100]mm/sec CNT100;
   1:  PR[91,1] = PR[90,1] + 19.532;
   1:  PR[91,2] = PR[90,2] + -17.979;
   1:L PR[91] R[100]mm/sec CNT100;
   1:  PR[91,1] = PR[90,1] + 20.627;
   1:  PR[91,2] = PR[90,2] + -18.173;
   1:L PR[91] R[100]mm/sec CNT100;
   1:  PR[91,1] = PR[90,1] + 22.487;
   1:  PR[91,2] = PR[90,2] + -18.321;
   1:L PR[91] R[100]mm/sec CNT100;
   1:  PR[91,1] = PR[90,1] + 25.513;
   1:  PR[91,2] = PR[90,2] + -18.133;
   1:L PR[91] R[100]mm/sec CNT100;
   1:  PR[91,1] = PR[90,1] + 27.391;
   1:  PR[91,2] = PR[90,2] + -17.738;
   1:L PR[91] R[100]mm/sec CNT100;
   1:  PR[91,1] = PR[90,1] + 28.313;
   1:  PR[91,2] = PR[90,2] + -17.463;
   1:L PR[91] R[100]mm/sec CNT100;
   1:  PR[91,1] = PR[90,1] + 30.176;
   1:  PR[91,2] = PR[90,2] + -16.781;
   1:L PR[91] R[100]mm/sec CNT100;
   1:  PR[91,1] = PR[90,1] + 31.958;
   1:  PR[91,2] = PR[90,2] + -15.820;
   1:L PR[91] R[100]mm/sec CNT100;
   1:  PR[91,1] = PR[90,1] + 32.755;
   1:  PR[91,2] = PR[90,2] + -15.362;
   1:L PR[91] R[100]mm/sec CNT100;
   1:  PR[91,1] = PR[90,1] + 34.319;
   1:  PR[91,2] = PR[90,2] + -14.201;
   1:L PR[91] R[100]mm/sec CNT100;
   1:  PR[91,1] = PR[90,1] + 35.823;
   1:  PR[91,2] = PR[90,2] + -12.709;
   1:L PR[91] R[100]mm/sec CNT100;
   1:  PR[91,1] = PR[90,1] + 36.465;
   1:  PR[91,2] = PR[90,2] + -12.105;
   1:L PR[91] R[100]mm/sec CNT100;
   1:  PR[91,1] = PR[90,1] + 37.670;
   1:  PR[91,2] = PR[90,2] + -10.505;
   1:L PR[91] R[100]mm/sec CNT100;
   1:  PR[91,1] = PR[90,1] + 38.130;
   1:  PR[91,2] = PR[90,2] + -9.807;
   1:L PR[91] R[100]mm/sec CNT100;
   1:  PR[91,1] = PR[90,1] + 39.107;
   1:  PR[91,2] = PR[90,2] + -8.028;
   1:L PR[91] R[100]mm/sec CNT100;
   1:  PR[91,1] = PR[90,1] + 39.851;
   1:  PR[91,2] = PR[90,2] + -6.045;
   1:L PR[91] R[100]mm/sec CNT100;
   1:  PR[91,1] = PR[90,1] + 40.130;
   1:  PR[91,2] = PR[90,2] + -5.282;
   1:L PR[91] R[100]mm/sec CNT100;
   1:  PR[91,1] = PR[90,1] + 40.552;
   1:  PR[91,2] = PR[90,2] + -3.354;
   1:L PR[91] R[100]mm/sec CNT100;
   1:  PR[91,1] = PR[90,1] + 40.709;
   1:  PR[91,2] = PR[90,2] + -1.170;
   1:L PR[91] R[100]mm/sec CNT100;
   1:  PR[91,1] = PR[90,1] + 40.802;
   1:  PR[91,2] = PR[90,2] + -0.371;
   1:L PR[91] R[100]mm/sec CNT100;
   1:  PR[91,1] = PR[90,1] + 40.656;
   1:  PR[91,2] = PR[90,2] + 1.663;
   1:L PR[91] R[100]mm/sec CNT100;
   1:  PR[91,1] = PR[90,1] + 40.563;
   1:  PR[91,2] = PR[90,2] + 2.455;
   1:L PR[91] R[100]mm/sec CNT100;
   1:  PR[91,1] = PR[90,1] + 40.132;
   1:  PR[91,2] = PR[90,2] + 4.428;
   1:L PR[91] R[100]mm/sec CNT100;
   1:  PR[91,1] = PR[90,1] + 39.106;
   1:  PR[91,2] = PR[90,2] + 7.183;
   1:L PR[91] R[100]mm/sec CNT100;
   1:  PR[91,1] = PR[90,1] + 38.130;
   1:  PR[91,2] = PR[90,2] + 8.960;
   1:L PR[91] R[100]mm/sec CNT100;
   1:  PR[91,1] = PR[90,1] + 37.670;
   1:  PR[91,2] = PR[90,2] + 9.657;
   1:L PR[91] R[100]mm/sec CNT100;
   1:  PR[91,1] = PR[90,1] + 36.446;
   1:  PR[91,2] = PR[90,2] + 11.282;
   1:L PR[91] R[100]mm/sec CNT100;
   1:  PR[91,1] = PR[90,1] + 34.971;
   1:  PR[91,2] = PR[90,2] + 12.746;
   1:L PR[91] R[100]mm/sec CNT100;
   1:  PR[91,1] = PR[90,1] + 34.345;
   1:  PR[91,2] = PR[90,2] + 13.335;
   1:L PR[91] R[100]mm/sec CNT100;
   1:  PR[91,1] = PR[90,1] + 32.781;
   1:  PR[91,2] = PR[90,2] + 14.495;
   1:L PR[91] R[100]mm/sec CNT100;
   1:  PR[91,1] = PR[90,1] + 30.914;
   1:  PR[91,2] = PR[90,2] + 15.501;
   1:L PR[91] R[100]mm/sec CNT100;
   1:  PR[91,1] = PR[90,1] + 30.144;
   1:  PR[91,2] = PR[90,2] + 15.945;
   1:L PR[91] R[100]mm/sec CNT100;
   1:  PR[91,1] = PR[90,1] + 28.314;
   1:  PR[91,2] = PR[90,2] + 16.615;
   1:L PR[91] R[100]mm/sec CNT100;
   1:  PR[91,1] = PR[90,1] + 27.391;
   1:  PR[91,2] = PR[90,2] + 16.890;
   1:L PR[91] R[100]mm/sec CNT100;
   1:  PR[91,1] = PR[90,1] + 25.513;
   1:  PR[91,2] = PR[90,2] + 17.286;
   1:L PR[91] R[100]mm/sec CNT100;
   1:  PR[91,1] = PR[90,1] + 22.488;
   1:  PR[91,2] = PR[90,2] + 17.473;
   1:L PR[91] R[100]mm/sec CNT100;
   1:  PR[91,1] = PR[90,1] + 20.627;
   1:  PR[91,2] = PR[90,2] + 17.325;
   1:L PR[91] R[100]mm/sec CNT100;
   1:  PR[91,1] = PR[90,1] + 19.532;
   1:  PR[91,2] = PR[90,2] + 17.132;
   1:L PR[91] R[100]mm/sec CNT100;
   1:  PR[91,1] = PR[90,1] + 17.706;
   1:  PR[91,2] = PR[90,2] + 16.718;
   1:L PR[91] R[100]mm/sec CNT100;
   1:  PR[91,1] = PR[90,1] + 15.949;
   1:  PR[91,2] = PR[90,2] + 16.044;
   1:L PR[91] R[100]mm/sec CNT100;
   1:  PR[91,1] = PR[90,1] + 14.872;
   1:  PR[91,2] = PR[90,2] + 15.580;
   1:L PR[91] R[100]mm/sec CNT100;
   1:  PR[91,1] = PR[90,1] + 13.339;
   1:  PR[91,2] = PR[90,2] + 14.722;
   1:L PR[91] R[100]mm/sec CNT100;
   1:  PR[91,1] = PR[90,1] + 11.832;
   1:  PR[91,2] = PR[90,2] + 13.568;
   1:L PR[91] R[100]mm/sec CNT100;
   1:  PR[91,1] = PR[90,1] + 10.841;
   1:  PR[91,2] = PR[90,2] + 12.833;
   1:L PR[91] R[100]mm/sec CNT100;
   1:  PR[91,1] = PR[90,1] + 9.637;
   1:  PR[91,2] = PR[90,2] + 11.601;
   1:L PR[91] R[100]mm/sec CNT100;
   1:  PR[91,1] = PR[90,1] + 8.775;
   1:  PR[91,2] = PR[90,2] + 10.575;
   1:L PR[91] R[100]mm/sec CNT100;
   1:  PR[91,1] = PR[90,1] + 7.769;
   1:  PR[91,2] = PR[90,2] + 9.196;
   1:L PR[91] R[100]mm/sec CNT100;
   1:  PR[91,1] = PR[90,1] + 6.943;
   1:  PR[91,2] = PR[90,2] + 7.634;
   1:L PR[91] R[100]mm/sec CNT100;
   1:  PR[91,1] = PR[90,1] + 6.324;
   1:  PR[91,2] = PR[90,2] + 6.414;
   1:L PR[91] R[100]mm/sec CNT100;
   1:  PR[91,1] = PR[90,1] + 6.174;
   1:  PR[91,2] = PR[90,2] + 5.993;
   1:L PR[91] R[100]mm/sec CNT100;
   1:  PR[91,1] = PR[90,1] + 7.064;
   1:  PR[91,2] = PR[90,2] + 4.899;
   1:L PR[91] R[100]mm/sec CNT100;
   1:  PR[91,1] = PR[90,1] + 5.113;
   1:  PR[91,2] = PR[90,2] + 3.702;
   1:L PR[91] R[100]mm/sec CNT100;
   1:  PR[91,1] = PR[90,1] + 4.431;
   1:  PR[91,2] = PR[90,2] + 2.593;
   1:L PR[91] R[100]mm/sec CNT100;
   1:  PR[91,1] = PR[90,1] + 2.200;
   1:  PR[91,2] = PR[90,2] + 1.767;
   1:L PR[91] R[100]mm/sec CNT100;
   1:  PR[91] = PR[90];
   1:  PR[91,1] = PR[90,1] + -2.705;
   1:  PR[91,2] = PR[90,2] + 2.312;
   1:  PR[91,3] = PR[90,3] + 7.995;
   1:L PR[91] R[100]mm/sec CNT100;
   1:  PR[91,1] = PR[90,1] + -4.685;
   1:  PR[91,2] = PR[90,2] + 3.057;
   1:L PR[91] R[100]mm/sec CNT100;
   1:  PR[91,1] = PR[90,1] + -5.659;
   1:  PR[91,2] = PR[90,2] + 4.120;
   1:L PR[91] R[100]mm/sec CNT100;
   1:  PR[91,1] = PR[90,1] + -6.177;
   1:  PR[91,2] = PR[90,2] + 4.924;
   1:L PR[91] R[100]mm/sec CNT100;
   1:  PR[91,1] = PR[90,1] + -6.513;
   1:  PR[91,2] = PR[90,2] + 5.889;
   1:L PR[91] R[100]mm/sec CNT100;
   1:  PR[91,1] = PR[90,1] + -6.869;
   1:  PR[91,2] = PR[90,2] + 6.562;
   1:L PR[91] R[100]mm/sec CNT100;
   1:  PR[91,1] = PR[90,1] + -8.252;
   1:  PR[91,2] = PR[90,2] + 9.349;
   1:L PR[91] R[100]mm/sec CNT100;
   1:  PR[91,1] = PR[90,1] + -8.721;
   1:  PR[91,2] = PR[90,2] + 9.992;
   1:L PR[91] R[100]mm/sec CNT100;
   1:  PR[91,1] = PR[90,1] + -10.482;
   1:  PR[91,2] = PR[90,2] + 12.088;
   1:L PR[91] R[100]mm/sec CNT100;
   1:  PR[91,1] = PR[90,1] + -11.113;
   1:  PR[91,2] = PR[90,2] + 12.734;
   1:L PR[91] R[100]mm/sec CNT100;
   1:  PR[91,1] = PR[90,1] + -11.888;
   1:  PR[91,2] = PR[90,2] + 13.327;
   1:L PR[91] R[100]mm/sec CNT100;
   1:  PR[91,1] = PR[90,1] + -13.999;
   1:  PR[91,2] = PR[90,2] + 14.894;
   1:L PR[91] R[100]mm/sec CNT100;
   1:  PR[91,1] = PR[90,1] + -14.812;
   1:  PR[91,2] = PR[90,2] + 15.349;
   1:L PR[91] R[100]mm/sec CNT100;
   1:  PR[91,1] = PR[90,1] + -15.871;
   1:  PR[91,2] = PR[90,2] + 15.756;
   1:L PR[91] R[100]mm/sec CNT100;
   1:  PR[91,1] = PR[90,1] + -18.180;
   1:  PR[91,2] = PR[90,2] + 16.747;
   1:L PR[91] R[100]mm/sec CNT100;
   1:  PR[91,1] = PR[90,1] + -19.231;
   1:  PR[91,2] = PR[90,2] + 16.985;
   1:L PR[91] R[100]mm/sec CNT100;
   1:  PR[91,1] = PR[90,1] + -21.496;
   1:  PR[91,2] = PR[90,2] + 17.385;
   1:L PR[91] R[100]mm/sec CNT100;
   1:  PR[91,1] = PR[90,1] + -22.657;
   1:  PR[91,2] = PR[90,2] + 17.477;
   1:L PR[91] R[100]mm/sec CNT100;
   1:  PR[91,1] = PR[90,1] + -26.113;
   1:  PR[91,2] = PR[90,2] + 17.268;
   1:L PR[91] R[100]mm/sec CNT100;
   1:  PR[91,1] = PR[90,1] + -27.340;
   1:  PR[91,2] = PR[90,2] + 17.010;
   1:L PR[91] R[100]mm/sec CNT100;
   1:  PR[91,1] = PR[90,1] + -29.269;
   1:  PR[91,2] = PR[90,2] + 16.435;
   1:L PR[91] R[100]mm/sec CNT100;
   1:  PR[91,1] = PR[90,1] + -30.539;
   1:  PR[91,2] = PR[90,2] + 15.969;
   1:L PR[91] R[100]mm/sec CNT100;
   1:  PR[91,1] = PR[90,1] + -31.766;
   1:  PR[91,2] = PR[90,2] + 15.308;
   1:L PR[91] R[100]mm/sec CNT100;
   1:  PR[91,1] = PR[90,1] + -33.439;
   1:  PR[91,2] = PR[90,2] + 14.345;
   1:L PR[91] R[100]mm/sec CNT100;
   1:  PR[91,1] = PR[90,1] + -34.520;
   1:  PR[91,2] = PR[90,2] + 13.544;
   1:L PR[91] R[100]mm/sec CNT100;
   1:  PR[91,1] = PR[90,1] + -35.596;
   1:  PR[91,2] = PR[90,2] + 12.476;
   1:L PR[91] R[100]mm/sec CNT100;
   1:  PR[91,1] = PR[90,1] + -36.948;
   1:  PR[91,2] = PR[90,2] + 11.203;
   1:L PR[91] R[100]mm/sec CNT100;
   1:  PR[91,1] = PR[90,1] + -37.804;
   1:  PR[91,2] = PR[90,2] + 10.067;
   1:L PR[91] R[100]mm/sec CNT100;
   1:  PR[91,1] = PR[90,1] + -38.777;
   1:  PR[91,2] = PR[90,2] + 8.591;
   1:L PR[91] R[100]mm/sec CNT100;
   1:  PR[91,1] = PR[90,1] + -39.479;
   1:  PR[91,2] = PR[90,2] + 7.312;
   1:L PR[91] R[100]mm/sec CNT100;
   1:  PR[91,1] = PR[90,1] + -40.620;
   1:  PR[91,2] = PR[90,2] + 4.229;
   1:L PR[91] R[100]mm/sec CNT100;
   1:  PR[91,1] = PR[90,1] + -40.922;
   1:  PR[91,2] = PR[90,2] + 2.849;
   1:L PR[91] R[100]mm/sec CNT100;
   1:  PR[91,1] = PR[90,1] + -41.039;
   1:  PR[91,2] = PR[90,2] + 1.221;
   1:L PR[91] R[100]mm/sec CNT100;
   1:  PR[91,1] = PR[90,1] + -41.237;
   1:  PR[91,2] = PR[90,2] + -0.477;
   1:L PR[91] R[100]mm/sec CNT100;
   1:  PR[91,1] = PR[90,1] + -41.130;
   1:  PR[91,2] = PR[90,2] + -1.963;
   1:L PR[91] R[100]mm/sec CNT100;
   1:  PR[91,1] = PR[90,1] + -40.933;
   1:  PR[91,2] = PR[90,2] + -3.644;
   1:L PR[91] R[100]mm/sec CNT100;
   1:  PR[91,1] = PR[90,1] + -40.620;
   1:  PR[91,2] = PR[90,2] + -5.077;
   1:L PR[91] R[100]mm/sec CNT100;
   1:  PR[91,1] = PR[90,1] + -39.479;
   1:  PR[91,2] = PR[90,2] + -8.159;
   1:L PR[91] R[100]mm/sec CNT100;
   1:  PR[91,1] = PR[90,1] + -38.776;
   1:  PR[91,2] = PR[90,2] + -9.438;
   1:L PR[91] R[100]mm/sec CNT100;
   1:  PR[91,1] = PR[90,1] + -37.803;
   1:  PR[91,2] = PR[90,2] + -10.915;
   1:L PR[91] R[100]mm/sec CNT100;
   1:  PR[91,1] = PR[90,1] + -36.929;
   1:  PR[91,2] = PR[90,2] + -12.076;
   1:L PR[91] R[100]mm/sec CNT100;
   1:  PR[91,1] = PR[90,1] + -35.866;
   1:  PR[91,2] = PR[90,2] + -13.130;
   1:L PR[91] R[100]mm/sec CNT100;
   1:  PR[91,1] = PR[90,1] + -34.545;
   1:  PR[91,2] = PR[90,2] + -14.372;
   1:L PR[91] R[100]mm/sec CNT100;
   1:  PR[91,1] = PR[90,1] + -33.465;
   1:  PR[91,2] = PR[90,2] + -15.173;
   1:L PR[91] R[100]mm/sec CNT100;
   1:  PR[91,1] = PR[90,1] + -32.128;
   1:  PR[91,2] = PR[90,2] + -15.894;
   1:L PR[91] R[100]mm/sec CNT100;
   1:  PR[91,1] = PR[90,1] + -30.506;
   1:  PR[91,2] = PR[90,2] + -16.829;
   1:L PR[91] R[100]mm/sec CNT100;
   1:  PR[91,1] = PR[90,1] + -29.267;
   1:  PR[91,2] = PR[90,2] + -17.282;
   1:L PR[91] R[100]mm/sec CNT100;
   1:  PR[91,1] = PR[90,1] + -27.338;
   1:  PR[91,2] = PR[90,2] + -17.857;
   1:L PR[91] R[100]mm/sec CNT100;
   1:  PR[91,1] = PR[90,1] + -26.111;
   1:  PR[91,2] = PR[90,2] + -18.115;
   1:L PR[91] R[100]mm/sec CNT100;
   1:  PR[91,1] = PR[90,1] + -22.655;
   1:  PR[91,2] = PR[90,2] + -18.324;
   1:L PR[91] R[100]mm/sec CNT100;
   1:  PR[91,1] = PR[90,1] + -21.494;
   1:  PR[91,2] = PR[90,2] + -18.232;
   1:L PR[91] R[100]mm/sec CNT100;
   1:  PR[91,1] = PR[90,1] + -19.229;
   1:  PR[91,2] = PR[90,2] + -17.831;
   1:L PR[91] R[100]mm/sec CNT100;
   1:  PR[91,1] = PR[90,1] + -18.131;
   1:  PR[91,2] = PR[90,2] + -17.583;
   1:L PR[91] R[100]mm/sec CNT100;
   1:  PR[91,1] = PR[90,1] + -17.072;
   1:  PR[91,2] = PR[90,2] + -17.176;
   1:L PR[91] R[100]mm/sec CNT100;
   1:  PR[91,1] = PR[90,1] + -14.852;
   1:  PR[91,2] = PR[90,2] + -16.219;
   1:L PR[91] R[100]mm/sec CNT100;
   1:  PR[91,1] = PR[90,1] + -14.011;
   1:  PR[91,2] = PR[90,2] + -15.749;
   1:L PR[91] R[100]mm/sec CNT100;
   1:  PR[91,1] = PR[90,1] + -13.134;
   1:  PR[91,2] = PR[90,2] + -15.077;
   1:L PR[91] R[100]mm/sec CNT100;
   1:  PR[91,1] = PR[90,1] + -11.098;
   1:  PR[91,2] = PR[90,2] + -13.566;
   1:L PR[91] R[100]mm/sec CNT100;
   1:  PR[91,1] = PR[90,1] + -10.480;
   1:  PR[91,2] = PR[90,2] + -12.933;
   1:L PR[91] R[100]mm/sec CNT100;
   1:  PR[91,1] = PR[90,1] + -8.719;
   1:  PR[91,2] = PR[90,2] + -10.836;
   1:L PR[91] R[100]mm/sec CNT100;
   1:  PR[91,1] = PR[90,1] + -8.231;
   1:  PR[91,2] = PR[90,2] + -10.167;
   1:L PR[91] R[100]mm/sec CNT100;
   1:  PR[91,1] = PR[90,1] + -7.816;
   1:  PR[91,2] = PR[90,2] + -9.382;
   1:L PR[91] R[100]mm/sec CNT100;
   1:  PR[91,1] = PR[90,1] + -6.562;
   1:  PR[91,2] = PR[90,2] + -6.906;
   1:L PR[91] R[100]mm/sec CNT100;
   1:  PR[91,1] = PR[90,1] + -5.981;
   1:  PR[91,2] = PR[90,2] + -5.235;
   1:L PR[91] R[100]mm/sec CNT100;
   1:  PR[91,1] = PR[90,1] + -5.500;
   1:  PR[91,2] = PR[90,2] + -4.939;
   1:L PR[91] R[100]mm/sec CNT100;
   1:  PR[91,1] = PR[90,1] + -4.915;
   1:  PR[91,2] = PR[90,2] + -3.989;
   1:L PR[91] R[100]mm/sec CNT100;
   1:  PR[91,1] = PR[90,1] + -2.695;
   1:  PR[91,2] = PR[90,2] + -3.159;
   1:L PR[91] R[100]mm/sec CNT100;
   1:  PR[91,1] = PR[90,1] + 2.234;
   1:L PR[91] R[100]mm/sec CNT100;
   1:  PR[91,1] = PR[90,1] + 4.209;
   1:  PR[91,2] = PR[90,2] + -3.907;
   1:L PR[91] R[100]mm/sec CNT100;
   1:  PR[91,1] = PR[90,1] + 5.185;
   1:  PR[91,2] = PR[90,2] + -4.976;
   1:L PR[91] R[100]mm/sec CNT100;
   1:  PR[91,1] = PR[90,1] + 5.698;
   1:  PR[91,2] = PR[90,2] + -5.771;
   1:L PR[91] R[100]mm/sec CNT100;
   1:  PR[91,1] = PR[90,1] + 6.027;
   1:  PR[91,2] = PR[90,2] + -6.716;
   1:L PR[91] R[100]mm/sec CNT100;
   1:  PR[91,1] = PR[90,1] + 6.374;
   1:  PR[91,2] = PR[90,2] + -7.372;
   1:L PR[91] R[100]mm/sec CNT100;
   1:  PR[91,1] = PR[90,1] + 7.772;
   1:  PR[91,2] = PR[90,2] + -10.194;
   1:L PR[91] R[100]mm/sec CNT100;
   1:  PR[91,1] = PR[90,1] + 8.241;
   1:  PR[91,2] = PR[90,2] + -10.837;
   1:L PR[91] R[100]mm/sec CNT100;
   1:  PR[91,1] = PR[90,1] + 10.002;
   1:  PR[91,2] = PR[90,2] + -12.935;
   1:L PR[91] R[100]mm/sec CNT100;
   1:  PR[91,1] = PR[90,1] + 10.632;
   1:  PR[91,2] = PR[90,2] + -13.580;
   1:L PR[91] R[100]mm/sec CNT100;
   1:  PR[91,1] = PR[90,1] + 11.407;
   1:  PR[91,2] = PR[90,2] + -14.173;
   1:L PR[91] R[100]mm/sec CNT100;
   1:  PR[91,1] = PR[90,1] + 13.518;
   1:  PR[91,2] = PR[90,2] + -15.741;
   1:L PR[91] R[100]mm/sec CNT100;
   1:  PR[91,1] = PR[90,1] + 14.331;
   1:  PR[91,2] = PR[90,2] + -16.196;
   1:L PR[91] R[100]mm/sec CNT100;
   1:  PR[91,1] = PR[90,1] + 15.390;
   1:  PR[91,2] = PR[90,2] + -16.602;
   1:L PR[91] R[100]mm/sec CNT100;
   1:  PR[91,1] = PR[90,1] + 17.699;
   1:  PR[91,2] = PR[90,2] + -17.593;
   1:L PR[91] R[100]mm/sec CNT100;
   1:  PR[91,1] = PR[90,1] + 18.750;
   1:  PR[91,2] = PR[90,2] + -17.832;
   1:L PR[91] R[100]mm/sec CNT100;
   1:  PR[91,1] = PR[90,1] + 21.016;
   1:  PR[91,2] = PR[90,2] + -18.232;
   1:L PR[91] R[100]mm/sec CNT100;
   1:  PR[91,1] = PR[90,1] + 22.176;
   1:  PR[91,2] = PR[90,2] + -18.324;
   1:L PR[91] R[100]mm/sec CNT100;
   1:  PR[91,1] = PR[90,1] + 25.633;
   1:  PR[91,2] = PR[90,2] + -18.115;
   1:L PR[91] R[100]mm/sec CNT100;
   1:  PR[91,1] = PR[90,1] + 26.859;
   1:  PR[91,2] = PR[90,2] + -17.857;
   1:L PR[91] R[100]mm/sec CNT100;
   1:  PR[91,1] = PR[90,1] + 28.788;
   1:  PR[91,2] = PR[90,2] + -17.282;
   1:L PR[91] R[100]mm/sec CNT100;
   1:  PR[91,1] = PR[90,1] + 30.059;
   1:  PR[91,2] = PR[90,2] + -16.817;
   1:L PR[91] R[100]mm/sec CNT100;
   1:  PR[91,1] = PR[90,1] + 31.286;
   1:  PR[91,2] = PR[90,2] + -16.155;
   1:L PR[91] R[100]mm/sec CNT100;
   1:  PR[91,1] = PR[90,1] + 32.959;
   1:  PR[91,2] = PR[90,2] + -15.193;
   1:L PR[91] R[100]mm/sec CNT100;
   1:  PR[91,1] = PR[90,1] + 34.039;
   1:  PR[91,2] = PR[90,2] + -14.392;
   1:L PR[91] R[100]mm/sec CNT100;
   1:  PR[91,1] = PR[90,1] + 35.116;
   1:  PR[91,2] = PR[90,2] + -13.324;
   1:L PR[91] R[100]mm/sec CNT100;
   1:  PR[91,1] = PR[90,1] + 36.468;
   1:  PR[91,2] = PR[90,2] + -12.050;
   1:L PR[91] R[100]mm/sec CNT100;
   1:  PR[91,1] = PR[90,1] + 37.324;
   1:  PR[91,2] = PR[90,2] + -10.914;
   1:L PR[91] R[100]mm/sec CNT100;
   1:  PR[91,1] = PR[90,1] + 38.297;
   1:  PR[91,2] = PR[90,2] + -9.438;
   1:L PR[91] R[100]mm/sec CNT100;
   1:  PR[91,1] = PR[90,1] + 39.002;
   1:  PR[91,2] = PR[90,2] + -8.154;
   1:L PR[91] R[100]mm/sec CNT100;
   1:  PR[91,1] = PR[90,1] + 39.546;
   1:  PR[91,2] = PR[90,2] + -6.702;
   1:L PR[91] R[100]mm/sec CNT100;
   1:  PR[91,1] = PR[90,1] + 40.140;
   1:  PR[91,2] = PR[90,2] + -5.082;
   1:L PR[91] R[100]mm/sec CNT100;
   1:  PR[91,1] = PR[90,1] + 40.442;
   1:  PR[91,2] = PR[90,2] + -3.698;
   1:L PR[91] R[100]mm/sec CNT100;
   1:  PR[91,1] = PR[90,1] + 40.559;
   1:  PR[91,2] = PR[90,2] + -2.069;
   1:L PR[91] R[100]mm/sec CNT100;
   1:  PR[91,1] = PR[90,1] + 40.757;
   1:  PR[91,2] = PR[90,2] + -0.371;
   1:L PR[91] R[100]mm/sec CNT100;
   1:  PR[91,1] = PR[90,1] + 40.650;
   1:  PR[91,2] = PR[90,2] + 1.116;
   1:L PR[91] R[100]mm/sec CNT100;
   1:  PR[91,1] = PR[90,1] + 40.454;
   1:  PR[91,2] = PR[90,2] + 2.798;
   1:L PR[91] R[100]mm/sec CNT100;
   1:  PR[91,1] = PR[90,1] + 40.141;
   1:  PR[91,2] = PR[90,2] + 4.230;
   1:L PR[91] R[100]mm/sec CNT100;
   1:  PR[91,1] = PR[90,1] + 38.999;
   1:  PR[91,2] = PR[90,2] + 7.311;
   1:L PR[91] R[100]mm/sec CNT100;
   1:  PR[91,1] = PR[90,1] + 38.297;
   1:  PR[91,2] = PR[90,2] + 8.591;
   1:L PR[91] R[100]mm/sec CNT100;
   1:  PR[91,1] = PR[90,1] + 37.324;
   1:  PR[91,2] = PR[90,2] + 10.066;
   1:L PR[91] R[100]mm/sec CNT100;
   1:  PR[91,1] = PR[90,1] + 36.449;
   1:  PR[91,2] = PR[90,2] + 11.228;
   1:L PR[91] R[100]mm/sec CNT100;
   1:  PR[91,1] = PR[90,1] + 35.387;
   1:  PR[91,2] = PR[90,2] + 12.282;
   1:L PR[91] R[100]mm/sec CNT100;
   1:  PR[91,1] = PR[90,1] + 34.065;
   1:  PR[91,2] = PR[90,2] + 13.525;
   1:L PR[91] R[100]mm/sec CNT100;
   1:  PR[91,1] = PR[90,1] + 32.986;
   1:  PR[91,2] = PR[90,2] + 14.326;
   1:L PR[91] R[100]mm/sec CNT100;
   1:  PR[91,1] = PR[90,1] + 31.649;
   1:  PR[91,2] = PR[90,2] + 15.047;
   1:L PR[91] R[100]mm/sec CNT100;
   1:  PR[91,1] = PR[90,1] + 30.027;
   1:  PR[91,2] = PR[90,2] + 15.981;
   1:L PR[91] R[100]mm/sec CNT100;
   1:  PR[91,1] = PR[90,1] + 28.789;
   1:  PR[91,2] = PR[90,2] + 16.435;
   1:L PR[91] R[100]mm/sec CNT100;
   1:  PR[91,1] = PR[90,1] + 26.860;
   1:  PR[91,2] = PR[90,2] + 17.010;
   1:L PR[91] R[100]mm/sec CNT100;
   1:  PR[91,1] = PR[90,1] + 25.633;
   1:  PR[91,2] = PR[90,2] + 17.268;
   1:L PR[91] R[100]mm/sec CNT100;
   1:  PR[91,1] = PR[90,1] + 22.177;
   1:  PR[91,2] = PR[90,2] + 17.477;
   1:L PR[91] R[100]mm/sec CNT100;
   1:  PR[91,1] = PR[90,1] + 21.016;
   1:  PR[91,2] = PR[90,2] + 17.385;
   1:L PR[91] R[100]mm/sec CNT100;
   1:  PR[91,1] = PR[90,1] + 18.751;
   1:  PR[91,2] = PR[90,2] + 16.985;
   1:L PR[91] R[100]mm/sec CNT100;
   1:  PR[91,1] = PR[90,1] + 17.654;
   1:  PR[91,2] = PR[90,2] + 16.736;
   1:L PR[91] R[100]mm/sec CNT100;
   1:  PR[91,1] = PR[90,1] + 16.594;
   1:  PR[91,2] = PR[90,2] + 16.329;
   1:L PR[91] R[100]mm/sec CNT100;
   1:  PR[91,1] = PR[90,1] + 14.374;
   1:  PR[91,2] = PR[90,2] + 15.373;
   1:L PR[91] R[100]mm/sec CNT100;
   1:  PR[91,1] = PR[90,1] + 13.534;
   1:  PR[91,2] = PR[90,2] + 14.903;
   1:L PR[91] R[100]mm/sec CNT100;
   1:  PR[91,1] = PR[90,1] + 12.656;
   1:  PR[91,2] = PR[90,2] + 14.231;
   1:L PR[91] R[100]mm/sec CNT100;
   1:  PR[91,1] = PR[90,1] + 10.620;
   1:  PR[91,2] = PR[90,2] + 12.721;
   1:L PR[91] R[100]mm/sec CNT100;
   1:  PR[91,1] = PR[90,1] + 10.003;
   1:  PR[91,2] = PR[90,2] + 12.088;
   1:L PR[91] R[100]mm/sec CNT100;
   1:  PR[91,1] = PR[90,1] + 8.242;
   1:  PR[91,2] = PR[90,2] + 9.990;
   1:L PR[91] R[100]mm/sec CNT100;
   1:  PR[91,1] = PR[90,1] + 7.754;
   1:  PR[91,2] = PR[90,2] + 9.322;
   1:L PR[91] R[100]mm/sec CNT100;
   1:  PR[91,1] = PR[90,1] + 7.338;
   1:  PR[91,2] = PR[90,2] + 8.537;
   1:L PR[91] R[100]mm/sec CNT100;
   1:  PR[91,1] = PR[90,1] + 6.080;
   1:  PR[91,2] = PR[90,2] + 6.055;
   1:L PR[91] R[100]mm/sec CNT100;
   1:  PR[91,1] = PR[90,1] + 5.501;
   1:  PR[91,2] = PR[90,2] + 4.386;
   1:L PR[91] R[100]mm/sec CNT100;
   1:  PR[91,1] = PR[90,1] + 5.020;
   1:  PR[91,2] = PR[90,2] + 4.091;
   1:L PR[91] R[100]mm/sec CNT100;
   1:  PR[91,1] = PR[90,1] + 4.436;
   1:  PR[91,2] = PR[90,2] + 3.143;
   1:L PR[91] R[100]mm/sec CNT100;
   1:  PR[91,1] = PR[90,1] + 2.221;
   1:  PR[91,2] = PR[90,2] + 2.312;
   1:L PR[91] R[100]mm/sec CNT100;
   1:  PR[91] = PR[90];
   1:  PR[91,1] = PR[90,1] + -2.729;
   1:  PR[91,2] = PR[90,2] + 2.856;
   1:  PR[91,3] = PR[90,3] + 9.295;
   1:L PR[91] R[100]mm/sec CNT100;
   1:  PR[91,1] = PR[90,1] + -4.744;
   1:  PR[91,2] = PR[90,2] + 3.626;
   1:L PR[91] R[100]mm/sec CNT100;
   1:  PR[91,1] = PR[90,1] + -5.312;
   1:  PR[91,2] = PR[90,2] + 4.304;
   1:L PR[91] R[100]mm/sec CNT100;
   1:  PR[91,1] = PR[90,1] + -6.036;
   1:  PR[91,2] = PR[90,2] + 5.064;
   1:L PR[91] R[100]mm/sec CNT100;
   1:  PR[91,1] = PR[90,1] + -8.225;
   1:  PR[91,2] = PR[90,2] + 9.453;
   1:L PR[91] R[100]mm/sec CNT100;
   1:  PR[91,1] = PR[90,1] + -10.848;
   1:  PR[91,2] = PR[90,2] + 12.576;
   1:L PR[91] R[100]mm/sec CNT100;
   1:  PR[91,1] = PR[90,1] + -10.893;
   1:  PR[91,2] = PR[90,2] + 12.622;
   1:L PR[91] R[100]mm/sec CNT100;
   1:  PR[91,1] = PR[90,1] + -11.001;
   1:  PR[91,2] = PR[90,2] + 12.705;
   1:L PR[91] R[100]mm/sec CNT100;
   1:  PR[91,1] = PR[90,1] + -14.194;
   1:  PR[91,2] = PR[90,2] + 15.075;
   1:L PR[91] R[100]mm/sec CNT100;
   1:  PR[91,1] = PR[90,1] + -14.315;
   1:  PR[91,2] = PR[90,2] + 15.143;
   1:L PR[91] R[100]mm/sec CNT100;
   1:  PR[91,1] = PR[90,1] + -14.633;
   1:  PR[91,2] = PR[90,2] + 15.265;
   1:L PR[91] R[100]mm/sec CNT100;
   1:  PR[91,1] = PR[90,1] + -18.127;
   1:  PR[91,2] = PR[90,2] + 16.765;
   1:L PR[91] R[100]mm/sec CNT100;
   1:  PR[91,1] = PR[90,1] + -18.450;
   1:  PR[91,2] = PR[90,2] + 16.838;
   1:L PR[91] R[100]mm/sec CNT100;
   1:  PR[91,1] = PR[90,1] + -21.885;
   1:  PR[91,2] = PR[90,2] + 17.444;
   1:L PR[91] R[100]mm/sec CNT100;
   1:  PR[91,1] = PR[90,1] + -22.346;
   1:  PR[91,2] = PR[90,2] + 17.480;
   1:L PR[91] R[100]mm/sec CNT100;
   1:  PR[91,1] = PR[90,1] + -26.233;
   1:  PR[91,2] = PR[90,2] + 17.250;
   1:L PR[91] R[100]mm/sec CNT100;
   1:  PR[91,1] = PR[90,1] + -26.808;
   1:  PR[91,2] = PR[90,2] + 17.129;
   1:L PR[91] R[100]mm/sec CNT100;
   1:  PR[91,1] = PR[90,1] + -29.743;
   1:  PR[91,2] = PR[90,2] + 16.254;
   1:L PR[91] R[100]mm/sec CNT100;
   1:  PR[91,1] = PR[90,1] + -30.423;
   1:  PR[91,2] = PR[90,2] + 16.005;
   1:L PR[91] R[100]mm/sec CNT100;
   1:  PR[91,1] = PR[90,1] + -31.095;
   1:  PR[91,2] = PR[90,2] + 15.642;
   1:L PR[91] R[100]mm/sec CNT100;
   1:  PR[91,1] = PR[90,1] + -33.643;
   1:  PR[91,2] = PR[90,2] + 14.176;
   1:L PR[91] R[100]mm/sec CNT100;
   1:  PR[91,1] = PR[90,1] + -34.240;
   1:  PR[91,2] = PR[90,2] + 13.734;
   1:L PR[91] R[100]mm/sec CNT100;
   1:  PR[91,1] = PR[90,1] + -34.889;
   1:  PR[91,2] = PR[90,2] + 13.090;
   1:L PR[91] R[100]mm/sec CNT100;
   1:  PR[91,1] = PR[90,1] + -36.952;
   1:  PR[91,2] = PR[90,2] + 11.148;
   1:L PR[91] R[100]mm/sec CNT100;
   1:  PR[91,1] = PR[90,1] + -37.458;
   1:  PR[91,2] = PR[90,2] + 10.476;
   1:L PR[91] R[100]mm/sec CNT100;
   1:  PR[91,1] = PR[90,1] + -38.943;
   1:  PR[91,2] = PR[90,2] + 8.222;
   1:L PR[91] R[100]mm/sec CNT100;
   1:  PR[91,1] = PR[90,1] + -39.373;
   1:  PR[91,2] = PR[90,2] + 7.440;
   1:L PR[91] R[100]mm/sec CNT100;
   1:  PR[91,1] = PR[90,1] + -40.629;
   1:  PR[91,2] = PR[90,2] + 4.030;
   1:L PR[91] R[100]mm/sec CNT100;
   1:  PR[91,1] = PR[90,1] + -40.813;
   1:  PR[91,2] = PR[90,2] + 3.192;
   1:L PR[91] R[100]mm/sec CNT100;
   1:  PR[91,1] = PR[90,1] + -40.890;
   1:  PR[91,2] = PR[90,2] + 2.119;
   1:L PR[91] R[100]mm/sec CNT100;
   1:  PR[91,1] = PR[90,1] + -41.192;
   1:  PR[91,2] = PR[90,2] + -0.477;
   1:L PR[91] R[100]mm/sec CNT100;
   1:  PR[91,1] = PR[90,1] + -41.124;
   1:  PR[91,2] = PR[90,2] + -1.416;
   1:L PR[91] R[100]mm/sec CNT100;
   1:  PR[91,1] = PR[90,1] + -40.824;
   1:  PR[91,2] = PR[90,2] + -3.988;
   1:L PR[91] R[100]mm/sec CNT100;
   1:  PR[91,1] = PR[90,1] + -40.629;
   1:  PR[91,2] = PR[90,2] + -4.878;
   1:L PR[91] R[100]mm/sec CNT100;
   1:  PR[91,1] = PR[90,1] + -39.373;
   1:  PR[91,2] = PR[90,2] + -8.288;
   1:L PR[91] R[100]mm/sec CNT100;
   1:  PR[91,1] = PR[90,1] + -38.943;
   1:  PR[91,2] = PR[90,2] + -9.069;
   1:L PR[91] R[100]mm/sec CNT100;
   1:  PR[91,1] = PR[90,1] + -37.457;
   1:  PR[91,2] = PR[90,2] + -11.324;
   1:L PR[91] R[100]mm/sec CNT100;
   1:  PR[91,1] = PR[90,1] + -36.932;
   1:  PR[91,2] = PR[90,2] + -12.021;
   1:L PR[91] R[100]mm/sec CNT100;
   1:  PR[91,1] = PR[90,1] + -36.281;
   1:  PR[91,2] = PR[90,2] + -12.667;
   1:L PR[91] R[100]mm/sec CNT100;
   1:  PR[91,1] = PR[90,1] + -34.265;
   1:  PR[91,2] = PR[90,2] + -14.563;
   1:L PR[91] R[100]mm/sec CNT100;
   1:  PR[91,1] = PR[90,1] + -33.669;
   1:  PR[91,2] = PR[90,2] + -15.005;
   1:L PR[91] R[100]mm/sec CNT100;
   1:  PR[91,1] = PR[90,1] + -32.862;
   1:  PR[91,2] = PR[90,2] + -15.440;
   1:L PR[91] R[100]mm/sec CNT100;
   1:  PR[91,1] = PR[90,1] + -30.389;
   1:  PR[91,2] = PR[90,2] + -16.865;
   1:L PR[91] R[100]mm/sec CNT100;
   1:  PR[91,1] = PR[90,1] + -29.742;
   1:  PR[91,2] = PR[90,2] + -17.102;
   1:L PR[91] R[100]mm/sec CNT100;
   1:  PR[91,1] = PR[90,1] + -26.806;
   1:  PR[91,2] = PR[90,2] + -17.977;
   1:L PR[91] R[100]mm/sec CNT100;
   1:  PR[91,1] = PR[90,1] + -26.230;
   1:  PR[91,2] = PR[90,2] + -18.098;
   1:L PR[91] R[100]mm/sec CNT100;
   1:  PR[91,1] = PR[90,1] + -22.343;
   1:  PR[91,2] = PR[90,2] + -18.327;
   1:L PR[91] R[100]mm/sec CNT100;
   1:  PR[91,1] = PR[90,1] + -21.882;
   1:  PR[91,2] = PR[90,2] + -18.291;
   1:L PR[91] R[100]mm/sec CNT100;
   1:  PR[91,1] = PR[90,1] + -18.446;
   1:  PR[91,2] = PR[90,2] + -17.684;
   1:L PR[91] R[100]mm/sec CNT100;
   1:  PR[91,1] = PR[90,1] + -18.077;
   1:  PR[91,2] = PR[90,2] + -17.600;
   1:L PR[91] R[100]mm/sec CNT100;
   1:  PR[91,1] = PR[90,1] + -17.716;
   1:  PR[91,2] = PR[90,2] + -17.462;
   1:L PR[91] R[100]mm/sec CNT100;
   1:  PR[91,1] = PR[90,1] + -14.353;
   1:  PR[91,2] = PR[90,2] + -16.011;
   1:L PR[91] R[100]mm/sec CNT100;
   1:  PR[91,1] = PR[90,1] + -14.191;
   1:  PR[91,2] = PR[90,2] + -15.920;
   1:L PR[91] R[100]mm/sec CNT100;
   1:  PR[91,1] = PR[90,1] + -10.878;
   1:  PR[91,2] = PR[90,2] + -13.453;
   1:L PR[91] R[100]mm/sec CNT100;
   1:  PR[91,1] = PR[90,1] + -10.845;
   1:  PR[91,2] = PR[90,2] + -13.420;
   1:L PR[91] R[100]mm/sec CNT100;
   1:  PR[91,1] = PR[90,1] + -8.217;
   1:  PR[91,2] = PR[90,2] + -10.289;
   1:L PR[91] R[100]mm/sec CNT100;
   1:  PR[91,1] = PR[90,1] + -6.313;
   1:  PR[91,2] = PR[90,2] + -6.538;
   1:L PR[91] R[100]mm/sec CNT100;
   1:  PR[91,1] = PR[90,1] + -6.025;
   1:  PR[91,2] = PR[90,2] + -5.708;
   1:L PR[91] R[100]mm/sec CNT100;
   1:  PR[91,1] = PR[90,1] + -5.407;
   1:  PR[91,2] = PR[90,2] + -5.329;
   1:L PR[91] R[100]mm/sec CNT100;
   1:  PR[91,1] = PR[90,1] + -4.920;
   1:  PR[91,2] = PR[90,2] + -4.537;
   1:L PR[91] R[100]mm/sec CNT100;
   1:  PR[91,1] = PR[90,1] + -2.711;
   1:  PR[91,2] = PR[90,2] + -3.703;
   1:L PR[91] R[100]mm/sec CNT100;
   1:  PR[91,1] = PR[90,1] + 2.302;
   1:L PR[91] R[100]mm/sec CNT100;
   1:  PR[91,1] = PR[90,1] + 3.047;
   1:  PR[91,2] = PR[90,2] + -4.016;
   1:L PR[91] R[100]mm/sec CNT100;
   1:  PR[91,1] = PR[90,1] + 4.247;
   1:  PR[91,2] = PR[90,2] + -4.459;
   1:L PR[91] R[100]mm/sec CNT100;
   1:  PR[91,1] = PR[90,1] + 4.741;
   1:  PR[91,2] = PR[90,2] + -5.040;
   1:L PR[91] R[100]mm/sec CNT100;
   1:  PR[91,1] = PR[90,1] + 4.790;
   1:  PR[91,2] = PR[90,2] + -5.081;
   1:L PR[91] R[100]mm/sec CNT100;
   1:  PR[91,1] = PR[90,1] + 5.559;
   1:  PR[91,2] = PR[90,2] + -5.927;
   1:L PR[91] R[100]mm/sec CNT100;
   1:  PR[91,1] = PR[90,1] + 6.264;
   1:  PR[91,2] = PR[90,2] + -7.307;
   1:L PR[91] R[100]mm/sec CNT100;
   1:  PR[91,1] = PR[90,1] + 7.745;
   1:  PR[91,2] = PR[90,2] + -10.298;
   1:L PR[91] R[100]mm/sec CNT100;
   1:  PR[91,1] = PR[90,1] + 10.367;
   1:  PR[91,2] = PR[90,2] + -13.422;
   1:L PR[91] R[100]mm/sec CNT100;
   1:  PR[91,1] = PR[90,1] + 10.411;
   1:  PR[91,2] = PR[90,2] + -13.467;
   1:L PR[91] R[100]mm/sec CNT100;
   1:  PR[91,1] = PR[90,1] + 10.520;
   1:  PR[91,2] = PR[90,2] + -13.551;
   1:L PR[91] R[100]mm/sec CNT100;
   1:  PR[91,1] = PR[90,1] + 13.712;
   1:  PR[91,2] = PR[90,2] + -15.921;
   1:L PR[91] R[100]mm/sec CNT100;
   1:  PR[91,1] = PR[90,1] + 13.833;
   1:  PR[91,2] = PR[90,2] + -15.989;
   1:L PR[91] R[100]mm/sec CNT100;
   1:  PR[91,1] = PR[90,1] + 14.151;
   1:  PR[91,2] = PR[90,2] + -16.111;
   1:L PR[91] R[100]mm/sec CNT100;
   1:  PR[91,1] = PR[90,1] + 17.646;
   1:  PR[91,2] = PR[90,2] + -17.611;
   1:L PR[91] R[100]mm/sec CNT100;
   1:  PR[91,1] = PR[90,1] + 17.969;
   1:  PR[91,2] = PR[90,2] + -17.684;
   1:L PR[91] R[100]mm/sec CNT100;
   1:  PR[91,1] = PR[90,1] + 21.404;
   1:  PR[91,2] = PR[90,2] + -18.291;
   1:L PR[91] R[100]mm/sec CNT100;
   1:  PR[91,1] = PR[90,1] + 21.865;
   1:  PR[91,2] = PR[90,2] + -18.328;
   1:L PR[91] R[100]mm/sec CNT100;
   1:  PR[91,1] = PR[90,1] + 25.752;
   1:  PR[91,2] = PR[90,2] + -18.098;
   1:L PR[91] R[100]mm/sec CNT100;
   1:  PR[91,1] = PR[90,1] + 26.328;
   1:  PR[91,2] = PR[90,2] + -17.976;
   1:L PR[91] R[100]mm/sec CNT100;
   1:  PR[91,1] = PR[90,1] + 29.263;
   1:  PR[91,2] = PR[90,2] + -17.102;
   1:L PR[91] R[100]mm/sec CNT100;
   1:  PR[91,1] = PR[90,1] + 29.942;
   1:  PR[91,2] = PR[90,2] + -16.853;
   1:L PR[91] R[100]mm/sec CNT100;
   1:  PR[91,1] = PR[90,1] + 30.614;
   1:  PR[91,2] = PR[90,2] + -16.490;
   1:L PR[91] R[100]mm/sec CNT100;
   1:  PR[91,1] = PR[90,1] + 33.163;
   1:  PR[91,2] = PR[90,2] + -15.024;
   1:L PR[91] R[100]mm/sec CNT100;
   1:  PR[91,1] = PR[90,1] + 33.760;
   1:  PR[91,2] = PR[90,2] + -14.582;
   1:L PR[91] R[100]mm/sec CNT100;
   1:  PR[91,1] = PR[90,1] + 34.409;
   1:  PR[91,2] = PR[90,2] + -13.938;
   1:L PR[91] R[100]mm/sec CNT100;
   1:  PR[91,1] = PR[90,1] + 36.471;
   1:  PR[91,2] = PR[90,2] + -11.995;
   1:L PR[91] R[100]mm/sec CNT100;
   1:  PR[91,1] = PR[90,1] + 36.978;
   1:  PR[91,2] = PR[90,2] + -11.323;
   1:L PR[91] R[100]mm/sec CNT100;
   1:  PR[91,1] = PR[90,1] + 38.464;
   1:  PR[91,2] = PR[90,2] + -9.069;
   1:L PR[91] R[100]mm/sec CNT100;
   1:  PR[91,1] = PR[90,1] + 38.896;
   1:  PR[91,2] = PR[90,2] + -8.281;
   1:L PR[91] R[100]mm/sec CNT100;
   1:  PR[91,1] = PR[90,1] + 39.242;
   1:  PR[91,2] = PR[90,2] + -7.358;
   1:L PR[91] R[100]mm/sec CNT100;
   1:  PR[91,1] = PR[90,1] + 40.149;
   1:  PR[91,2] = PR[90,2] + -4.882;
   1:L PR[91] R[100]mm/sec CNT100;
   1:  PR[91,1] = PR[90,1] + 40.333;
   1:  PR[91,2] = PR[90,2] + -4.042;
   1:L PR[91] R[100]mm/sec CNT100;
   1:  PR[91,1] = PR[90,1] + 40.410;
   1:  PR[91,2] = PR[90,2] + -2.968;
   1:L PR[91] R[100]mm/sec CNT100;
   1:  PR[91,1] = PR[90,1] + 40.712;
   1:  PR[91,2] = PR[90,2] + -0.370;
   1:L PR[91] R[100]mm/sec CNT100;
   1:  PR[91,1] = PR[90,1] + 40.645;
   1:  PR[91,2] = PR[90,2] + 0.569;
   1:L PR[91] R[100]mm/sec CNT100;
   1:  PR[91,1] = PR[90,1] + 40.344;
   1:  PR[91,2] = PR[90,2] + 3.142;
   1:L PR[91] R[100]mm/sec CNT100;
   1:  PR[91,1] = PR[90,1] + 40.150;
   1:  PR[91,2] = PR[90,2] + 4.032;
   1:L PR[91] R[100]mm/sec CNT100;
   1:  PR[91,1] = PR[90,1] + 38.893;
   1:  PR[91,2] = PR[90,2] + 7.439;
   1:L PR[91] R[100]mm/sec CNT100;
   1:  PR[91,1] = PR[90,1] + 38.464;
   1:  PR[91,2] = PR[90,2] + 8.221;
   1:L PR[91] R[100]mm/sec CNT100;
   1:  PR[91,1] = PR[90,1] + 36.978;
   1:  PR[91,2] = PR[90,2] + 10.476;
   1:L PR[91] R[100]mm/sec CNT100;
   1:  PR[91,1] = PR[90,1] + 36.453;
   1:  PR[91,2] = PR[90,2] + 11.173;
   1:L PR[91] R[100]mm/sec CNT100;
   1:  PR[91,1] = PR[90,1] + 35.802;
   1:  PR[91,2] = PR[90,2] + 11.818;
   1:L PR[91] R[100]mm/sec CNT100;
   1:  PR[91,1] = PR[90,1] + 33.786;
   1:  PR[91,2] = PR[90,2] + 13.715;
   1:L PR[91] R[100]mm/sec CNT100;
   1:  PR[91,1] = PR[90,1] + 33.190;
   1:  PR[91,2] = PR[90,2] + 14.157;
   1:L PR[91] R[100]mm/sec CNT100;
   1:  PR[91,1] = PR[90,1] + 32.383;
   1:  PR[91,2] = PR[90,2] + 14.592;
   1:L PR[91] R[100]mm/sec CNT100;
   1:  PR[91,1] = PR[90,1] + 29.911;
   1:  PR[91,2] = PR[90,2] + 16.017;
   1:L PR[91] R[100]mm/sec CNT100;
   1:  PR[91,1] = PR[90,1] + 29.264;
   1:  PR[91,2] = PR[90,2] + 16.254;
   1:L PR[91] R[100]mm/sec CNT100;
   1:  PR[91,1] = PR[90,1] + 26.328;
   1:  PR[91,2] = PR[90,2] + 17.129;
   1:L PR[91] R[100]mm/sec CNT100;
   1:  PR[91,1] = PR[90,1] + 25.747;
   1:  PR[91,2] = PR[90,2] + 17.251;
   1:L PR[91] R[100]mm/sec CNT100;
   1:  PR[91,1] = PR[90,1] + 25.063;
   1:  PR[91,2] = PR[90,2] + 17.295;
   1:L PR[91] R[100]mm/sec CNT100;
   1:  PR[91,1] = PR[90,1] + 21.868;
   1:  PR[91,2] = PR[90,2] + 17.481;
   1:L PR[91] R[100]mm/sec CNT100;
   1:  PR[91,1] = PR[90,1] + 21.405;
   1:  PR[91,2] = PR[90,2] + 17.444;
   1:L PR[91] R[100]mm/sec CNT100;
   1:  PR[91,1] = PR[90,1] + 17.970;
   1:  PR[91,2] = PR[90,2] + 16.837;
   1:L PR[91] R[100]mm/sec CNT100;
   1:  PR[91,1] = PR[90,1] + 17.601;
   1:  PR[91,2] = PR[90,2] + 16.754;
   1:L PR[91] R[100]mm/sec CNT100;
   1:  PR[91,1] = PR[90,1] + 17.239;
   1:  PR[91,2] = PR[90,2] + 16.615;
   1:L PR[91] R[100]mm/sec CNT100;
   1:  PR[91,1] = PR[90,1] + 13.877;
   1:  PR[91,2] = PR[90,2] + 15.166;
   1:L PR[91] R[100]mm/sec CNT100;
   1:  PR[91,1] = PR[90,1] + 13.714;
   1:  PR[91,2] = PR[90,2] + 15.075;
   1:L PR[91] R[100]mm/sec CNT100;
   1:  PR[91,1] = PR[90,1] + 10.401;
   1:  PR[91,2] = PR[90,2] + 12.610;
   1:L PR[91] R[100]mm/sec CNT100;
   1:  PR[91,1] = PR[90,1] + 10.368;
   1:  PR[91,2] = PR[90,2] + 12.576;
   1:L PR[91] R[100]mm/sec CNT100;
   1:  PR[91,1] = PR[90,1] + 7.740;
   1:  PR[91,2] = PR[90,2] + 9.445;
   1:L PR[91] R[100]mm/sec CNT100;
   1:  PR[91,1] = PR[90,1] + 5.831;
   1:  PR[91,2] = PR[90,2] + 5.685;
   1:L PR[91] R[100]mm/sec CNT100;
   1:  PR[91,1] = PR[90,1] + 5.545;
   1:  PR[91,2] = PR[90,2] + 4.860;
   1:L PR[91] R[100]mm/sec CNT100;
   1:  PR[91,1] = PR[90,1] + 4.927;
   1:  PR[91,2] = PR[90,2] + 4.481;
   1:L PR[91] R[100]mm/sec CNT100;
   1:  PR[91,1] = PR[90,1] + 4.442;
   1:  PR[91,2] = PR[90,2] + 3.692;
   1:L PR[91] R[100]mm/sec CNT100;
   1:  PR[91,1] = PR[90,1] + 2.242;
   1:  PR[91,2] = PR[90,2] + 2.856;
   1:L PR[91] R[100]mm/sec CNT100;
   1:  PR[91] = PR[90];
   1:  PR[91,1] = PR[90,1] + -2.754;
   1:  PR[91,2] = PR[90,2] + 3.401;
   1:  PR[91,3] = PR[90,3] + 10.595;
   1:L PR[91] R[100]mm/sec CNT100;
   1:  PR[91,1] = PR[90,1] + -4.751;
   1:  PR[91,2] = PR[90,2] + 4.176;
   1:L PR[91] R[100]mm/sec CNT100;
   1:  PR[91,1] = PR[90,1] + -5.298;
   1:  PR[91,2] = PR[90,2] + 4.828;
   1:L PR[91] R[100]mm/sec CNT100;
   1:  PR[91,1] = PR[90,1] + -5.329;
   1:  PR[91,2] = PR[90,2] + 4.853;
   1:L PR[91] R[100]mm/sec CNT100;
   1:  PR[91,1] = PR[90,1] + -5.978;
   1:  PR[91,2] = PR[90,2] + 5.553;
   1:L PR[91] R[100]mm/sec CNT100;
   1:  PR[91,1] = PR[90,1] + -7.680;
   1:  PR[91,2] = PR[90,2] + 8.902;
   1:L PR[91] R[100]mm/sec CNT100;
   1:  PR[91,1] = PR[90,1] + -8.130;
   1:  PR[91,2] = PR[90,2] + 9.643;
   1:L PR[91] R[100]mm/sec CNT100;
   1:  PR[91,1] = PR[90,1] + -10.407;
   1:  PR[91,2] = PR[90,2] + 12.314;
   1:L PR[91] R[100]mm/sec CNT100;
   1:  PR[91,1] = PR[90,1] + -10.817;
   1:  PR[91,2] = PR[90,2] + 12.731;
   1:L PR[91] R[100]mm/sec CNT100;
   1:  PR[91,1] = PR[90,1] + -13.911;
   1:  PR[91,2] = PR[90,2] + 14.994;
   1:L PR[91] R[100]mm/sec CNT100;
   1:  PR[91,1] = PR[90,1] + -14.150;
   1:  PR[91,2] = PR[90,2] + 15.146;
   1:L PR[91] R[100]mm/sec CNT100;
   1:  PR[91,1] = PR[90,1] + -17.973;
   1:  PR[91,2] = PR[90,2] + 16.763;
   1:L PR[91] R[100]mm/sec CNT100;
   1:  PR[91,1] = PR[90,1] + -22.107;
   1:  PR[91,2] = PR[90,2] + 17.475;
   1:L PR[91] R[100]mm/sec CNT100;
   1:  PR[91,1] = PR[90,1] + -26.326;
   1:  PR[91,2] = PR[90,2] + 17.234;
   1:L PR[91] R[100]mm/sec CNT100;
   1:  PR[91,1] = PR[90,1] + -30.219;
   1:  PR[91,2] = PR[90,2] + 16.073;
   1:L PR[91] R[100]mm/sec CNT100;
   1:  PR[91,1] = PR[90,1] + -30.277;
   1:  PR[91,2] = PR[90,2] + 16.052;
   1:L PR[91] R[100]mm/sec CNT100;
   1:  PR[91,1] = PR[90,1] + -33.850;
   1:  PR[91,2] = PR[90,2] + 14.006;
   1:L PR[91] R[100]mm/sec CNT100;
   1:  PR[91,1] = PR[90,1] + -33.961;
   1:  PR[91,2] = PR[90,2] + 13.924;
   1:L PR[91] R[100]mm/sec CNT100;
   1:  PR[91,1] = PR[90,1] + -34.182;
   1:  PR[91,2] = PR[90,2] + 13.704;
   1:L PR[91] R[100]mm/sec CNT100;
   1:  PR[91,1] = PR[90,1] + -36.955;
   1:  PR[91,2] = PR[90,2] + 11.093;
   1:L PR[91] R[100]mm/sec CNT100;
   1:  PR[91,1] = PR[90,1] + -37.112;
   1:  PR[91,2] = PR[90,2] + 10.885;
   1:L PR[91] R[100]mm/sec CNT100;
   1:  PR[91,1] = PR[90,1] + -39.110;
   1:  PR[91,2] = PR[90,2] + 7.852;
   1:L PR[91] R[100]mm/sec CNT100;
   1:  PR[91,1] = PR[90,1] + -39.267;
   1:  PR[91,2] = PR[90,2] + 7.567;
   1:L PR[91] R[100]mm/sec CNT100;
